LIN {X 0,Y 354.791,Z 411.293,A -85,B 0,C 180,E1 -13362.867,E2 -13362.867} C_VEL
LIN {X 0,Y 354.834,Z 411.311,A -85,B 0,C 180,E1 -13366.661,E2 -13366.661} C_VEL
LIN {X 0,Y 355.442,Z 414.83,A -85,B 0,C 180,E1 -13369.27,E2 -13369.27} C_VEL
LIN {X 0,Y 356.124,Z 419.11,A -85,B 0,C 180,E1 -13372.282,E2 -13372.282} C_VEL
LIN {X 0,Y 356.314,Z 421.652,A -85,B 0,C 180,E1 -13373.968,E2 -13373.968} C_VEL
LIN {X 0,Y 356.012,Z 425.546,A -85,B 0,C 180,E1 -13376.444,E2 -13376.444} C_VEL
LIN {X 0,Y 355.387,Z 431.994,A -85,B 0,C 180,E1 -13380.37,E2 -13380.37} C_VEL
LIN {X 0,Y 354.742,Z 438.379,A -85,B 0,C 180,E1 -13384.16,E2 -13384.16} C_VEL
LIN {X 0,Y 354.299,Z 444.723,A -85,B 0,C 180,E1 -13387.859,E2 -13387.859} C_VEL
LIN {X 0,Y 354.107,Z 447.535,A -85,B 0,C 180,E1 -13389.487,E2 -13389.487} C_VEL
LIN {X 0,Y 357.033,Z 461.918,A -85,B 0,C 180,E1 -13390.207,E2 -13390.207} C_VEL
LIN {X 0,Y 359.043,Z 475.173,A -85,B 0,C 180,E1 -13391.077,E2 -13391.077} C_VEL
LIN {X 0,Y 359.866,Z 484.104,A -85,B 0,C 180,E1 -13391.792,E2 -13391.792} C_VEL
LIN {X 0,Y 358.903,Z 495.118,A -85,B 0,C 180,E1 -13392.772,E2 -13392.772} C_VEL
LIN {X 0,Y 357.705,Z 506.362,A -85,B 0,C 180,E1 -13394.034,E2 -13394.034} C_VEL
LIN {X 0,Y 356.623,Z 516.327,A -85,B 0,C 180,E1 -13395.447,E2 -13395.447} C_VEL
LIN {X 0,Y 355.526,Z 525.99,A -85,B 0,C 180,E1 -13397.15,E2 -13397.15} C_VEL
LIN {X 0,Y 354.584,Z 533.681,A -85,B 0,C 180,E1 -13398.857,E2 -13398.857} C_VEL
LIN {X 0,Y 353.901,Z 540.779,A -85,B 0,C 180,E1 -13400.859,E2 -13400.859} C_VEL
LIN {X 0,Y 353.519,Z 545.502,A -85,B 0,C 180,E1 -13402.575,E2 -13402.575} C_VEL
LIN {X 0,Y 353.282,Z 549.111,A -85,B 0,C 180,E1 -13404.291,E2 -13404.291} C_VEL
LIN {X 0,Y 353.28,Z 550.976,A -85,B 0,C 180,E1 -13405.436,E2 -13405.436} C_VEL
LIN {X 0,Y 353.223,Z 552.372,A -85,B 0,C 180,E1 -13406.578,E2 -13406.578} C_VEL
LIN {X 0,Y 353.216,Z 553.978,A -85,B 0,C 180,E1 -13408.86,E2 -13408.86} C_VEL
LIN {X 0,Y 353.262,Z 554.194,A -85,B 0,C 180,E1 -13410,E2 -13410} C_VEL
LIN {X 0,Y 353.216,Z 553.974,A -85,B 0,C 180,E1 -13411.14,E2 -13411.14} C_VEL
LIN {X 0,Y 353.223,Z 552.364,A -85,B 0,C 180,E1 -13413.422,E2 -13413.422} C_VEL
LIN {X 0,Y 353.28,Z 550.964,A -85,B 0,C 180,E1 -13414.564,E2 -13414.564} C_VEL
LIN {X 0,Y 353.278,Z 548.719,A -85,B 0,C 180,E1 -13415.908,E2 -13415.908} C_VEL
LIN {X 0,Y 353.628,Z 544.039,A -85,B 0,C 180,E1 -13417.997,E2 -13417.997} C_VEL
LIN {X 0,Y 354.174,Z 537.919,A -85,B 0,C 180,E1 -13419.999,E2 -13419.999} C_VEL
LIN {X 0,Y 354.849,Z 531.235,A -85,B 0,C 180,E1 -13421.713,E2 -13421.713} C_VEL
LIN {X 0,Y 355.9,Z 522.95,A -85,B 0,C 180,E1 -13423.416,E2 -13423.416} C_VEL
LIN {X 0,Y 356.879,Z 514.454,A -85,B 0,C 180,E1 -13424.833,E2 -13424.833} C_VEL
LIN {X 0,Y 357.91,Z 503.953,A -85,B 0,C 180,E1 -13426.249,E2 -13426.249} C_VEL
LIN {X 0,Y 359.204,Z 492.142,A -85,B 0,C 180,E1 -13427.507,E2 -13427.507} C_VEL
LIN {X 0,Y 359.788,Z 482.88,A -85,B 0,C 180,E1 -13428.301,E2 -13428.301} C_VEL
LIN {X 0,Y 358.509,Z 471.103,A -85,B 0,C 180,E1 -13429.203,E2 -13429.203} C_VEL
LIN {X 0,Y 356.25,Z 457.832,A -85,B 0,C 180,E1 -13430.004,E2 -13430.004} C_VEL
LIN {X 0,Y 354.106,Z 447.512,A -85,B 0,C 180,E1 -13430.513,E2 -13430.513} C_VEL
LIN {X 0,Y 354.519,Z 441.111,A -85,B 0,C 180,E1 -13434.23,E2 -13434.23} C_VEL
LIN {X 0,Y 355.177,Z 434.088,A -85,B 0,C 180,E1 -13438.353,E2 -13438.353} C_VEL
LIN {X 0,Y 355.747,Z 428.287,A -85,B 0,C 180,E1 -13441.843,E2 -13441.843} C_VEL
LIN {X 0,Y 356.245,Z 423.356,A -85,B 0,C 180,E1 -13444.898,E2 -13444.898} C_VEL
LIN {X 0,Y 356.112,Z 418.838,A -85,B 0,C 180,E1 -13447.869,E2 -13447.869} C_VEL
LIN {X 0,Y 355.332,Z 414.036,A -85,B 0,C 180,E1 -13451.272,E2 -13451.272} C_VEL
LIN {X 0,Y 354.825,Z 411.291,A -85,B 0,C 180,E1 -13453.436,E2 -13453.436} C_VEL
LIN {X 0,Y 354.795,Z 411.288,A -85,B 0,C 180,E1 -13457.663,E2 -13457.663} C_VEL
LIN {X 0,Y 354.816,Z 411.287,A -85,B 0,C 180,E1 -13460.666,E2 -13460.666} C_VEL
LIN {X 0,Y 354.823,Z 411.285,A -85,B 0,C 180,E1 -13464.301,E2 -13464.301} C_VEL
LIN {X 0,Y 354.788,Z 411.288,A -85,B 0,C 180,E1 -13467.667,E2 -13467.667} C_VEL
LIN {X 0,Y 354.847,Z 411.28,A -85,B 0,C 180,E1 -13471.619,E2 -13471.619} C_VEL
LIN {X 0,Y 354.9,Z 411.275,A -85,B 0,C 180,E1 -13474.173,E2 -13474.173} C_VEL
LIN {X 0,Y 354.836,Z 411.282,A -85,B 0,C 180,E1 -13477.894,E2 -13477.894} C_VEL
LIN {X 0,Y 354.923,Z 411.271,A -85,B 0,C 180,E1 -13481.892,E2 -13481.892} C_VEL
LIN {X 0,Y 354.945,Z 411.27,A -85,B 0,C 180,E1 -13485.981,E2 -13485.981} C_VEL
LIN {X 0,Y 354.984,Z 411.264,A -85,B 0,C 180,E1 -13489.736,E2 -13489.736} C_VEL
LIN {X 0,Y 355.116,Z 411.25,A -85,B 0,C 180,E1 -13492.037,E2 -13492.037} C_VEL
LIN {X 0,Y 355.094,Z 411.256,A -85,B 0,C 180,E1 -13494.321,E2 -13494.321} C_VEL
LIN {X 0,Y 355.245,Z 411.232,A -85,B 0,C 180,E1 -13497.732,E2 -13497.732} C_VEL
LIN {X 0,Y 355.399,Z 411.215,A -85,B 0,C 180,E1 -13500,E2 -13500} C_VEL
LIN {X 0,Y 355.245,Z 411.236,A -85,B 0,C 180,E1 -13502.268,E2 -13502.268} C_VEL
LIN {X 0,Y 355.14,Z 411.244,A -85,B 0,C 180,E1 -13506.819,E2 -13506.819} C_VEL
LIN {X 0,Y 355.018,Z 411.259,A -85,B 0,C 180,E1 -13509.112,E2 -13509.112} C_VEL
LIN {X 0,Y 354.928,Z 411.271,A -85,B 0,C 180,E1 -13512.581,E2 -13512.581} C_VEL
LIN {X 0,Y 354.892,Z 411.279,A -85,B 0,C 180,E1 -13516.096,E2 -13516.096} C_VEL
LIN {X 0,Y 354.903,Z 411.274,A -85,B 0,C 180,E1 -13518.472,E2 -13518.472} C_VEL
LIN {X 0,Y 354.836,Z 411.285,A -85,B 0,C 180,E1 -13522.106,E2 -13522.106} C_VEL
LIN {X 0,Y 354.9,Z 411.279,A -85,B 0,C 180,E1 -13525.827,E2 -13525.827} C_VEL
LIN {X 0,Y 354.847,Z 411.286,A -85,B 0,C 180,E1 -13529.679,E2 -13529.679} C_VEL
LIN {X 0,Y 354.807,Z 411.29,A -85,B 0,C 180,E1 -13533.702,E2 -13533.702} C_VEL
LIN {X 0,Y 354.803,Z 411.286,A -85,B 0,C 180,E1 -13536.459,E2 -13536.459} C_VEL
LIN {X 0,Y 354.825,Z 411.289,A -85,B 0,C 180,E1 -13539.424,E2 -13539.424} C_VEL
LIN {X 0,Y 354.79,Z 411.289,A -85,B 0,C 180,E1 -13542.867,E2 -13542.867} C_VEL
LIN {X 0,Y 354.783,Z 411.289,A -85,B 0,C 180,E1 -13546.106,E2 -13546.106} C_VEL
LIN {X 0,Y 354.79,Z 411.293,A -85,B 0,C 180,E1 -13549.179,E2 -13549.179} C_VEL
LIN {X 0,Y 354.785,Z 411.293,A -85,B 0,C 180,E1 -13552.408,E2 -13552.408} C_VEL
LIN {X 0,Y 354.713,Z 411.303,A -85,B 0,C 180,E1 -13553.53,E2 -13553.53} C_VEL
LIN {X 0,Y 354.711,Z 414.22,A -85,B 0,C 180,E1 -13556.322,E2 -13556.322} C_VEL
LIN {X 0,Y 354.543,Z 417.115,A -85,B 0,C 180,E1 -13558.977,E2 -13558.977} C_VEL
LIN {X 0,Y 354.277,Z 421.498,A -85,B 0,C 180,E1 -13562.854,E2 -13562.854} C_VEL
LIN {X 0,Y 354.011,Z 425.915,A -85,B 0,C 180,E1 -13566.606,E2 -13566.606} C_VEL
LIN {X 0,Y 353.886,Z 429.701,A -85,B 0,C 180,E1 -13569.579,E2 -13569.579} C_VEL
LIN {X 0,Y 357.361,Z 443.1,A -85,B 0,C 180,E1 -13570.31,E2 -13570.31} C_VEL
LIN {X 0,Y 359.992,Z 455.598,A -85,B 0,C 180,E1 -13571.186,E2 -13571.186} C_VEL
LIN {X 0,Y 360.819,Z 460.678,A -85,B 0,C 180,E1 -13571.599,E2 -13571.599} C_VEL
LIN {X 0,Y 359.861,Z 471.979,A -85,B 0,C 180,E1 -13572.526,E2 -13572.526} C_VEL
LIN {X 0,Y 358.845,Z 482.845,A -85,B 0,C 180,E1 -13573.673,E2 -13573.673} C_VEL
LIN {X 0,Y 357.895,Z 492.362,A -85,B 0,C 180,E1 -13574.919,E2 -13574.919} C_VEL
LIN {X 0,Y 356.749,Z 501.204,A -85,B 0,C 180,E1 -13576.326,E2 -13576.326} C_VEL
LIN {X 0,Y 355.757,Z 509.824,A -85,B 0,C 180,E1 -13578.028,E2 -13578.028} C_VEL
LIN {X 0,Y 354.916,Z 516.695,A -85,B 0,C 180,E1 -13579.734,E2 -13579.734} C_VEL
LIN {X 0,Y 354.205,Z 522.198,A -85,B 0,C 180,E1 -13581.442,E2 -13581.442} C_VEL
LIN {X 0,Y 353.808,Z 526.852,A -85,B 0,C 180,E1 -13583.313,E2 -13583.313} C_VEL
LIN {X 0,Y 353.498,Z 530.652,A -85,B 0,C 180,E1 -13585.439,E2 -13585.439} C_VEL
LIN {X 0,Y 353.339,Z 532.051,A -85,B 0,C 180,E1 -13586.579,E2 -13586.579} C_VEL
LIN {X 0,Y 353.256,Z 533.656,A -85,B 0,C 180,E1 -13588.86,E2 -13588.86} C_VEL
LIN {X 0,Y 353.265,Z 533.887,A -85,B 0,C 180,E1 -13590,E2 -13590} C_VEL
LIN {X 0,Y 353.256,Z 533.698,A -85,B 0,C 180,E1 -13591.14,E2 -13591.14} C_VEL
LIN {X 0,Y 353.334,Z 532.147,A -85,B 0,C 180,E1 -13593.421,E2 -13593.421} C_VEL
LIN {X 0,Y 353.491,Z 530.789,A -85,B 0,C 180,E1 -13594.561,E2 -13594.561} C_VEL
LIN {X 0,Y 353.762,Z 527.213,A -85,B 0,C 180,E1 -13596.622,E2 -13596.622} C_VEL
LIN {X 0,Y 354.201,Z 522.482,A -85,B 0,C 180,E1 -13598.558,E2 -13598.558} C_VEL
LIN {X 0,Y 354.994,Z 516.044,A -85,B 0,C 180,E1 -13600.552,E2 -13600.552} C_VEL
LIN {X 0,Y 355.783,Z 508.972,A -85,B 0,C 180,E1 -13602.26,E2 -13602.26} C_VEL
LIN {X 0,Y 356.925,Z 500.154,A -85,B 0,C 180,E1 -13603.958,E2 -13603.958} C_VEL
LIN {X 0,Y 358.06,Z 491.103,A -85,B 0,C 180,E1 -13605.366,E2 -13605.366} C_VEL
LIN {X 0,Y 358.921,Z 481.466,A -85,B 0,C 180,E1 -13606.597,E2 -13606.597} C_VEL
LIN {X 0,Y 360.084,Z 469.933,A -85,B 0,C 180,E1 -13607.756,E2 -13607.756} C_VEL
LIN {X 0,Y 360.798,Z 460.4,A -85,B 0,C 180,E1 -13608.526,E2 -13608.526} C_VEL
LIN {X 0,Y 358.493,Z 448.093,A -85,B 0,C 180,E1 -13609.468,E2 -13609.468} C_VEL
LIN {X 0,Y 355.478,Z 435.673,A -85,B 0,C 180,E1 -13610.23,E2 -13610.23} C_VEL
LIN {X 0,Y 353.87,Z 429.539,A -85,B 0,C 180,E1 -13610.558,E2 -13610.558} C_VEL
LIN {X 0,Y 354.103,Z 424.577,A -85,B 0,C 180,E1 -13614.633,E2 -13614.633} C_VEL
LIN {X 0,Y 354.281,Z 421.637,A -85,B 0,C 180,E1 -13617.146,E2 -13617.146} C_VEL
LIN {X 0,Y 354.538,Z 417.231,A -85,B 0,C 180,E1 -13621.024,E2 -13621.024} C_VEL
LIN {X 0,Y 354.713,Z 414.326,A -85,B 0,C 180,E1 -13623.695,E2 -13623.695} C_VEL
LIN {X 0,Y 354.754,Z 411.408,A -85,B 0,C 180,E1 -13626.465,E2 -13626.465} C_VEL
LIN {X 0,Y 354.793,Z 411.291,A -85,B 0,C 180,E1 -13627.872,E2 -13627.872} C_VEL
LIN {X 0,Y 354.144,Z 411.374,A -85,B 0,C 180,E1 -13628.819,E2 -13628.819} C_VEL
LIN {X 0,Y 351.269,Z 411.728,A -85,B 0,C 180,E1 -13630.359,E2 -13630.359} C_VEL
LIN {X 0,Y 348.827,Z 412.03,A -85,B 0,C 180,E1 -13631.604,E2 -13631.604} C_VEL
LIN {X 0,Y 347.79,Z 412.163,A -85,B 0,C 180,E1 -13632.569,E2 -13632.569} C_VEL
LIN {X 0,Y 347.713,Z 412.167,A -85,B 0,C 180,E1 -13632.896,E2 -13632.896} C_VEL
LIN {X 0,Y 347.768,Z 412.165,A -85,B 0,C 180,E1 -13635.017,E2 -13635.017} C_VEL
LIN {X 0,Y 347.753,Z 412.168,A -85,B 0,C 180,E1 -13638.397,E2 -13638.397} C_VEL
LIN {X 0,Y 347.779,Z 412.162,A -85,B 0,C 180,E1 -13642.011,E2 -13642.011} C_VEL
LIN {X 0,Y 347.747,Z 412.165,A -85,B 0,C 180,E1 -13645.536,E2 -13645.536} C_VEL
LIN {X 0,Y 347.763,Z 412.163,A -85,B 0,C 180,E1 -13649.653,E2 -13649.653} C_VEL
LIN {X 0,Y 347.833,Z 412.154,A -85,B 0,C 180,E1 -13653.608,E2 -13653.608} C_VEL
LIN {X 0,Y 347.791,Z 412.164,A -85,B 0,C 180,E1 -13656.162,E2 -13656.162} C_VEL
LIN {X 0,Y 347.815,Z 412.159,A -85,B 0,C 180,E1 -13659.909,E2 -13659.909} C_VEL
LIN {X 0,Y 347.869,Z 412.154,A -85,B 0,C 180,E1 -13662.359,E2 -13662.359} C_VEL
LIN {X 0,Y 347.9,Z 412.15,A -85,B 0,C 180,E1 -13665.971,E2 -13665.971} C_VEL
LIN {X 0,Y 347.932,Z 412.143,A -85,B 0,C 180,E1 -13669.526,E2 -13669.526} C_VEL
LIN {X 0,Y 348.077,Z 412.128,A -85,B 0,C 180,E1 -13671.875,E2 -13671.875} C_VEL
LIN {X 0,Y 348.07,Z 412.128,A -85,B 0,C 180,E1 -13674.206,E2 -13674.206} C_VEL
LIN {X 0,Y 348.209,Z 412.111,A -85,B 0,C 180,E1 -13677.686,E2 -13677.686} C_VEL
LIN {X 0,Y 348.348,Z 412.094,A -85,B 0,C 180,E1 -13680,E2 -13680} C_VEL
LIN {X 0,Y 348.209,Z 412.108,A -85,B 0,C 180,E1 -13682.313,E2 -13682.313} C_VEL
LIN {X 0,Y 348.11,Z 412.12,A -85,B 0,C 180,E1 -13686.958,E2 -13686.958} C_VEL
LIN {X 0,Y 347.972,Z 412.14,A -85,B 0,C 180,E1 -13689.298,E2 -13689.298} C_VEL
LIN {X 0,Y 347.897,Z 412.147,A -85,B 0,C 180,E1 -13692.839,E2 -13692.839} C_VEL
LIN {X 0,Y 347.842,Z 412.153,A -85,B 0,C 180,E1 -13696.431,E2 -13696.431} C_VEL
LIN {X 0,Y 347.854,Z 412.153,A -85,B 0,C 180,E1 -13698.86,E2 -13698.86} C_VEL
LIN {X 0,Y 347.777,Z 412.161,A -85,B 0,C 180,E1 -13702.579,E2 -13702.579} C_VEL
LIN {X 0,Y 347.815,Z 412.16,A -85,B 0,C 180,E1 -13705.108,E2 -13705.108} C_VEL
LIN {X 0,Y 347.81,Z 412.159,A -85,B 0,C 180,E1 -13707.694,E2 -13707.694} C_VEL
LIN {X 0,Y 347.751,Z 412.165,A -85,B 0,C 180,E1 -13710.348,E2 -13710.348} C_VEL
LIN {X 0,Y 347.75,Z 412.164,A -85,B 0,C 180,E1 -13714.044,E2 -13714.044} C_VEL
LIN {X 0,Y 347.765,Z 412.166,A -85,B 0,C 180,E1 -13717.321,E2 -13717.321} C_VEL
LIN {X 0,Y 347.735,Z 412.168,A -85,B 0,C 180,E1 -13720.297,E2 -13720.297} C_VEL
LIN {X 0,Y 347.729,Z 412.172,A -85,B 0,C 180,E1 -13723.407,E2 -13723.407} C_VEL
LIN {X 0,Y 347.776,Z 412.228,A -85,B 0,C 180,E1 -13726.346,E2 -13726.346} C_VEL
LIN {X 0,Y 348.609,Z 417.085,A -85,B 0,C 180,E1 -13730.004,E2 -13730.004} C_VEL
LIN {X 0,Y 349.215,Z 421.12,A -85,B 0,C 180,E1 -13732.86,E2 -13732.86} C_VEL
LIN {X 0,Y 349.252,Z 424.325,A -85,B 0,C 180,E1 -13735.005,E2 -13735.005} C_VEL
LIN {X 0,Y 348.559,Z 430.751,A -85,B 0,C 180,E1 -13739.059,E2 -13739.059} C_VEL
LIN {X 0,Y 347.892,Z 436.757,A -85,B 0,C 180,E1 -13742.732,E2 -13742.732} C_VEL
LIN {X 0,Y 347.419,Z 442.433,A -85,B 0,C 180,E1 -13746.135,E2 -13746.135} C_VEL
LIN {X 0,Y 347.068,Z 447.32,A -85,B 0,C 180,E1 -13749.051,E2 -13749.051} C_VEL
LIN {X 0,Y 350.077,Z 461.716,A -85,B 0,C 180,E1 -13749.797,E2 -13749.797} C_VEL
LIN {X 0,Y 352.083,Z 474.968,A -85,B 0,C 180,E1 -13750.688,E2 -13750.688} C_VEL
LIN {X 0,Y 353.013,Z 485.675,A -85,B 0,C 180,E1 -13751.576,E2 -13751.576} C_VEL
LIN {X 0,Y 351.986,Z 496.339,A -85,B 0,C 180,E1 -13752.572,E2 -13752.572} C_VEL
LIN {X 0,Y 350.714,Z 507.306,A -85,B 0,C 180,E1 -13753.867,E2 -13753.867} C_VEL
LIN {X 0,Y 349.74,Z 516.125,A -85,B 0,C 180,E1 -13755.155,E2 -13755.155} C_VEL
LIN {X 0,Y 348.571,Z 525.787,A -85,B 0,C 180,E1 -13756.89,E2 -13756.89} C_VEL
LIN {X 0,Y 347.564,Z 533.477,A -85,B 0,C 180,E1 -13758.629,E2 -13758.629} C_VEL
LIN {X 0,Y 346.871,Z 540.575,A -85,B 0,C 180,E1 -13760.672,E2 -13760.672} C_VEL
LIN {X 0,Y 346.47,Z 545.298,A -85,B 0,C 180,E1 -13762.423,E2 -13762.423} C_VEL
LIN {X 0,Y 346.201,Z 548.907,A -85,B 0,C 180,E1 -13764.174,E2 -13764.174} C_VEL
LIN {X 0,Y 346.175,Z 550.771,A -85,B 0,C 180,E1 -13765.342,E2 -13765.342} C_VEL
LIN {X 0,Y 346.147,Z 552.169,A -85,B 0,C 180,E1 -13766.508,E2 -13766.508} C_VEL
LIN {X 0,Y 346.116,Z 553.774,A -85,B 0,C 180,E1 -13768.836,E2 -13768.836} C_VEL
LIN {X 0,Y 346.165,Z 553.99,A -85,B 0,C 180,E1 -13770,E2 -13770} C_VEL
LIN {X 0,Y 346.116,Z 553.769,A -85,B 0,C 180,E1 -13771.163,E2 -13771.163} C_VEL
LIN {X 0,Y 346.147,Z 552.16,A -85,B 0,C 180,E1 -13773.492,E2 -13773.492} C_VEL
LIN {X 0,Y 346.175,Z 550.759,A -85,B 0,C 180,E1 -13774.658,E2 -13774.658} C_VEL
LIN {X 0,Y 346.241,Z 547.814,A -85,B 0,C 180,E1 -13776.409,E2 -13776.409} C_VEL
LIN {X 0,Y 346.571,Z 543.833,A -85,B 0,C 180,E1 -13778.161,E2 -13778.161} C_VEL
LIN {X 0,Y 347.146,Z 537.713,A -85,B 0,C 180,E1 -13780.203,E2 -13780.203} C_VEL
LIN {X 0,Y 347.847,Z 531.028,A -85,B 0,C 180,E1 -13781.952,E2 -13781.952} C_VEL
LIN {X 0,Y 348.972,Z 522.743,A -85,B 0,C 180,E1 -13783.688,E2 -13783.688} C_VEL
LIN {X 0,Y 350.006,Z 514.247,A -85,B 0,C 180,E1 -13785.131,E2 -13785.131} C_VEL
LIN {X 0,Y 351.061,Z 503.745,A -85,B 0,C 180,E1 -13786.575,E2 -13786.575} C_VEL
LIN {X 0,Y 352.428,Z 491.934,A -85,B 0,C 180,E1 -13787.855,E2 -13787.855} C_VEL
LIN {X 0,Y 352.932,Z 483.739,A -85,B 0,C 180,E1 -13788.579,E2 -13788.579} C_VEL
LIN {X 0,Y 351.559,Z 470.884,A -85,B 0,C 180,E1 -13789.598,E2 -13789.598} C_VEL
LIN {X 0,Y 349.239,Z 457.562,A -85,B 0,C 180,E1 -13790.426,E2 -13790.426} C_VEL
LIN {X 0,Y 347.081,Z 447.329,A -85,B 0,C 180,E1 -13790.928,E2 -13790.928} C_VEL
LIN {X 0,Y 347.503,Z 441.37,A -85,B 0,C 180,E1 -13794.481,E2 -13794.481} C_VEL
LIN {X 0,Y 348.104,Z 434.977,A -85,B 0,C 180,E1 -13798.324,E2 -13798.324} C_VEL
LIN {X 0,Y 348.658,Z 429.637,A -85,B 0,C 180,E1 -13801.607,E2 -13801.607} C_VEL
LIN {X 0,Y 349.221,Z 424.267,A -85,B 0,C 180,E1 -13804.998,E2 -13804.998} C_VEL
LIN {X 0,Y 349.2,Z 421.046,A -85,B 0,C 180,E1 -13807.141,E2 -13807.141} C_VEL
LIN {X 0,Y 348.571,Z 416.771,A -85,B 0,C 180,E1 -13810.18,E2 -13810.18} C_VEL
LIN {X 0,Y 347.779,Z 412.169,A -85,B 0,C 180,E1 -13813.71,E2 -13813.71} C_VEL
LIN {X 0,Y 347.726,Z 412.172,A -85,B 0,C 180,E1 -13816.686,E2 -13816.686} C_VEL
LIN {X 0,Y 347.748,Z 412.166,A -85,B 0,C 180,E1 -13820.173,E2 -13820.173} C_VEL
LIN {X 0,Y 347.764,Z 412.167,A -85,B 0,C 180,E1 -13822.679,E2 -13822.679} C_VEL
LIN {X 0,Y 347.749,Z 412.165,A -85,B 0,C 180,E1 -13825.956,E2 -13825.956} C_VEL
LIN {X 0,Y 347.75,Z 412.165,A -85,B 0,C 180,E1 -13829.652,E2 -13829.652} C_VEL
LIN {X 0,Y 347.832,Z 412.154,A -85,B 0,C 180,E1 -13833.608,E2 -13833.608} C_VEL
LIN {X 0,Y 347.79,Z 412.161,A -85,B 0,C 180,E1 -13836.162,E2 -13836.162} C_VEL
LIN {X 0,Y 347.814,Z 412.157,A -85,B 0,C 180,E1 -13839.909,E2 -13839.909} C_VEL
LIN {X 0,Y 347.867,Z 412.154,A -85,B 0,C 180,E1 -13842.359,E2 -13842.359} C_VEL
LIN {X 0,Y 347.899,Z 412.147,A -85,B 0,C 180,E1 -13845.971,E2 -13845.971} C_VEL
LIN {X 0,Y 347.935,Z 412.142,A -85,B 0,C 180,E1 -13849.526,E2 -13849.526} C_VEL
LIN {X 0,Y 348.076,Z 412.125,A -85,B 0,C 180,E1 -13851.875,E2 -13851.875} C_VEL
LIN {X 0,Y 348.069,Z 412.129,A -85,B 0,C 180,E1 -13854.206,E2 -13854.206} C_VEL
LIN {X 0,Y 348.208,Z 412.108,A -85,B 0,C 180,E1 -13857.687,E2 -13857.687} C_VEL
LIN {X 0,Y 348.369,Z 412.091,A -85,B 0,C 180,E1 -13860,E2 -13860} C_VEL
LIN {X 0,Y 348.207,Z 412.112,A -85,B 0,C 180,E1 -13862.314,E2 -13862.314} C_VEL
LIN {X 0,Y 348.108,Z 412.12,A -85,B 0,C 180,E1 -13866.958,E2 -13866.958} C_VEL
LIN {X 0,Y 347.971,Z 412.137,A -85,B 0,C 180,E1 -13869.299,E2 -13869.299} C_VEL
LIN {X 0,Y 347.896,Z 412.146,A -85,B 0,C 180,E1 -13872.839,E2 -13872.839} C_VEL
LIN {X 0,Y 347.841,Z 412.155,A -85,B 0,C 180,E1 -13876.431,E2 -13876.431} C_VEL
LIN {X 0,Y 347.852,Z 412.151,A -85,B 0,C 180,E1 -13878.861,E2 -13878.861} C_VEL
LIN {X 0,Y 347.776,Z 412.161,A -85,B 0,C 180,E1 -13882.579,E2 -13882.579} C_VEL
LIN {X 0,Y 347.813,Z 412.157,A -85,B 0,C 180,E1 -13885.108,E2 -13885.108} C_VEL
LIN {X 0,Y 347.809,Z 412.163,A -85,B 0,C 180,E1 -13887.694,E2 -13887.694} C_VEL
LIN {X 0,Y 347.762,Z 412.163,A -85,B 0,C 180,E1 -13890.347,E2 -13890.347} C_VEL
LIN {X 0,Y 347.746,Z 412.165,A -85,B 0,C 180,E1 -13894.464,E2 -13894.464} C_VEL
LIN {X 0,Y 347.779,Z 412.163,A -85,B 0,C 180,E1 -13897.99,E2 -13897.99} C_VEL
LIN {X 0,Y 347.752,Z 412.166,A -85,B 0,C 180,E1 -13901.83,E2 -13901.83} C_VEL
LIN {X 0,Y 347.768,Z 412.165,A -85,B 0,C 180,E1 -13905.017,E2 -13905.017} C_VEL
LIN {X 0,Y 347.752,Z 412.165,A -85,B 0,C 180,E1 -13908.397,E2 -13908.397} C_VEL
LIN {X 0,Y 347.762,Z 412.168,A -85,B 0,C 180,E1 -13912.014,E2 -13912.014} C_VEL
LIN {X 0,Y 347.704,Z 412.733,A -85,B 0,C 180,E1 -13913.95,E2 -13913.95} C_VEL
LIN {X 0,Y 347.616,Z 415.827,A -85,B 0,C 180,E1 -13916.915,E2 -13916.915} C_VEL
LIN {X 0,Y 347.376,Z 419.657,A -85,B 0,C 180,E1 -13920.455,E2 -13920.455} C_VEL
LIN {X 0,Y 347.181,Z 423.157,A -85,B 0,C 180,E1 -13923.555,E2 -13923.555} C_VEL
LIN {X 0,Y 347.024,Z 426.109,A -85,B 0,C 180,E1 -13926.106,E2 -13926.106} C_VEL
LIN {X 0,Y 346.82,Z 429.857,A -85,B 0,C 180,E1 -13929.141,E2 -13929.141} C_VEL
LIN {X 0,Y 350.335,Z 443.072,A -85,B 0,C 180,E1 -13929.886,E2 -13929.886} C_VEL
LIN {X 0,Y 352.73,Z 454.179,A -85,B 0,C 180,E1 -13930.673,E2 -13930.673} C_VEL
LIN {X 0,Y 354.008,Z 462.099,A -85,B 0,C 180,E1 -13931.324,E2 -13931.324} C_VEL
LIN {X 0,Y 352.923,Z 473.628,A -85,B 0,C 180,E1 -13932.321,E2 -13932.321} C_VEL
LIN {X 0,Y 351.983,Z 483.625,A -85,B 0,C 180,E1 -13933.418,E2 -13933.418} C_VEL
LIN {X 0,Y 351.056,Z 492.569,A -85,B 0,C 180,E1 -13934.618,E2 -13934.618} C_VEL
LIN {X 0,Y 349.867,Z 501.411,A -85,B 0,C 180,E1 -13936.051,E2 -13936.051} C_VEL
LIN {X 0,Y 348.822,Z 510.03,A -85,B 0,C 180,E1 -13937.787,E2 -13937.787} C_VEL
LIN {X 0,Y 347.936,Z 516.901,A -85,B 0,C 180,E1 -13939.526,E2 -13939.526} C_VEL
LIN {X 0,Y 347.18,Z 522.403,A -85,B 0,C 180,E1 -13941.268,E2 -13941.268} C_VEL
LIN {X 0,Y 346.731,Z 527.351,A -85,B 0,C 180,E1 -13943.316,E2 -13943.316} C_VEL
LIN {X 0,Y 346.44,Z 530.856,A -85,B 0,C 180,E1 -13945.346,E2 -13945.346} C_VEL
LIN {X 0,Y 346.264,Z 532.255,A -85,B 0,C 180,E1 -13946.509,E2 -13946.509} C_VEL
LIN {X 0,Y 346.16,Z 533.86,A -85,B 0,C 180,E1 -13948.837,E2 -13948.837} C_VEL
LIN {X 0,Y 346.168,Z 534.091,A -85,B 0,C 180,E1 -13950,E2 -13950} C_VEL
LIN {X 0,Y 346.159,Z 533.901,A -85,B 0,C 180,E1 -13951.163,E2 -13951.163} C_VEL
LIN {X 0,Y 346.259,Z 532.35,A -85,B 0,C 180,E1 -13953.491,E2 -13953.491} C_VEL
LIN {X 0,Y 346.433,Z 530.992,A -85,B 0,C 180,E1 -13954.655,E2 -13954.655} C_VEL
LIN {X 0,Y 346.682,Z 527.715,A -85,B 0,C 180,E1 -13956.616,E2 -13956.616} C_VEL
LIN {X 0,Y 347.176,Z 522.685,A -85,B 0,C 180,E1 -13958.733,E2 -13958.733} C_VEL
LIN {X 0,Y 347.984,Z 516.247,A -85,B 0,C 180,E1 -13960.767,E2 -13960.767} C_VEL
LIN {X 0,Y 348.843,Z 509.174,A -85,B 0,C 180,E1 -13962.508,E2 -13962.508} C_VEL
LIN {X 0,Y 350.052,Z 500.354,A -85,B 0,C 180,E1 -13964.238,E2 -13964.238} C_VEL
LIN {X 0,Y 351.212,Z 491.419,A -85,B 0,C 180,E1 -13965.655,E2 -13965.655} C_VEL
LIN {X 0,Y 352.132,Z 481.665,A -85,B 0,C 180,E1 -13966.927,E2 -13966.927} C_VEL
LIN {X 0,Y 353.346,Z 470.131,A -85,B 0,C 180,E1 -13968.106,E2 -13968.106} C_VEL
LIN {X 0,Y 353.937,Z 460.879,A -85,B 0,C 180,E1 -13968.878,E2 -13968.878} C_VEL
LIN {X 0,Y 351.503,Z 448.297,A -85,B 0,C 180,E1 -13969.871,E2 -13969.871} C_VEL
LIN {X 0,Y 348.415,Z 435.647,A -85,B 0,C 180,E1 -13970.668,E2 -13970.668} C_VEL
LIN {X 0,Y 346.819,Z 429.759,A -85,B 0,C 180,E1 -13970.983,E2 -13970.983} C_VEL
LIN {X 0,Y 347.033,Z 425.753,A -85,B 0,C 180,E1 -13974.31,E2 -13974.31} C_VEL
LIN {X 0,Y 347.264,Z 421.813,A -85,B 0,C 180,E1 -13977.741,E2 -13977.741} C_VEL
LIN {X 0,Y 347.544,Z 417.398,A -85,B 0,C 180,E1 -13981.72,E2 -13981.72} C_VEL
LIN {X 0,Y 347.68,Z 414.472,A -85,B 0,C 180,E1 -13984.471,E2 -13984.471} C_VEL
LIN {X 0,Y 347.751,Z 412.838,A -85,B 0,C 180,E1 -13986.06,E2 -13986.06} C_VEL
LIN {X 0,Y 347.74,Z 412.17,A -85,B 0,C 180,E1 -13987.324,E2 -13987.324} C_VEL
LIN {X 0,Y 347.735,Z 412.168,A -85,B 0,C 180,E1 -13990.297,E2 -13990.297} C_VEL
LIN {X 0,Y 347.713,Z 412.167,A -85,B 0,C 180,E1 -13992.896,E2 -13992.896} C_VEL
LIN {X 0,Y 347.074,Z 412.25,A -85,B 0,C 180,E1 -13993.863,E2 -13993.863} C_VEL
LIN {X 0,Y 344.258,Z 412.601,A -85,B 0,C 180,E1 -13995.437,E2 -13995.437} C_VEL
LIN {X 0,Y 341.847,Z 412.906,A -85,B 0,C 180,E1 -13996.711,E2 -13996.711} C_VEL
LIN {X 0,Y 340.793,Z 413.032,A -85,B 0,C 180,E1 -13997.696,E2 -13997.696} C_VEL
LIN {X 0,Y 340.697,Z 413.044,A -85,B 0,C 180,E1 -13998.03,E2 -13998.03} C_VEL
LIN {X 0,Y 340.738,Z 413.038,A -85,B 0,C 180,E1 -14001.773,E2 -14001.773} C_VEL
LIN {X 0,Y 340.725,Z 413.04,A -85,B 0,C 180,E1 -14005.595,E2 -14005.595} C_VEL
LIN {X 0,Y 340.771,Z 413.036,A -85,B 0,C 180,E1 -14010.021,E2 -14010.021} C_VEL
LIN {X 0,Y 340.806,Z 413.03,A -85,B 0,C 180,E1 -14013.02,E2 -14013.02} C_VEL
LIN {X 0,Y 340.759,Z 413.036,A -85,B 0,C 180,E1 -14015.638,E2 -14015.638} C_VEL
LIN {X 0,Y 340.748,Z 413.037,A -85,B 0,C 180,E1 -14019.474,E2 -14019.474} C_VEL
LIN {X 0,Y 340.86,Z 413.027,A -85,B 0,C 180,E1 -14021.984,E2 -14021.984} C_VEL
LIN {X 0,Y 340.872,Z 413.023,A -85,B 0,C 180,E1 -14025.705,E2 -14025.705} C_VEL
LIN {X 0,Y 340.874,Z 413.021,A -85,B 0,C 180,E1 -14029.306,E2 -14029.306} C_VEL
LIN {X 0,Y 341.079,Z 412.996,A -85,B 0,C 180,E1 -14032.898,E2 -14032.898} C_VEL
LIN {X 0,Y 341.17,Z 412.988,A -85,B 0,C 180,E1 -14037.639,E2 -14037.639} C_VEL
LIN {X 0,Y 341.298,Z 412.973,A -85,B 0,C 180,E1 -14040,E2 -14040} C_VEL
LIN {X 0,Y 341.171,Z 412.985,A -85,B 0,C 180,E1 -14042.361,E2 -14042.361} C_VEL
LIN {X 0,Y 341.079,Z 412.997,A -85,B 0,C 180,E1 -14047.102,E2 -14047.102} C_VEL
LIN {X 0,Y 340.878,Z 413.02,A -85,B 0,C 180,E1 -14050.694,E2 -14050.694} C_VEL
LIN {X 0,Y 340.865,Z 413.022,A -85,B 0,C 180,E1 -14054.325,E2 -14054.325} C_VEL
LIN {X 0,Y 340.839,Z 413.025,A -85,B 0,C 180,E1 -14058.466,E2 -14058.466} C_VEL
LIN {X 0,Y 340.756,Z 413.037,A -85,B 0,C 180,E1 -14061.857,E2 -14061.857} C_VEL
LIN {X 0,Y 340.775,Z 413.036,A -85,B 0,C 180,E1 -14065.664,E2 -14065.664} C_VEL
LIN {X 0,Y 340.731,Z 413.039,A -85,B 0,C 180,E1 -14068.321,E2 -14068.321} C_VEL
LIN {X 0,Y 340.7,Z 413.047,A -85,B 0,C 180,E1 -14071.045,E2 -14071.045} C_VEL
LIN {X 0,Y 340.72,Z 413.044,A -85,B 0,C 180,E1 -14075.279,E2 -14075.279} C_VEL
LIN {X 0,Y 340.712,Z 413.042,A -85,B 0,C 180,E1 -14078.386,E2 -14078.386} C_VEL
LIN {X 0,Y 340.701,Z 413.044,A -85,B 0,C 180,E1 -14082.045,E2 -14082.045} C_VEL
LIN {X 0,Y 340.734,Z 413.105,A -85,B 0,C 180,E1 -14085.999,E2 -14085.999} C_VEL
LIN {X 0,Y 341.519,Z 417.738,A -85,B 0,C 180,E1 -14089.589,E2 -14089.589} C_VEL
LIN {X 0,Y 342.026,Z 420.957,A -85,B 0,C 180,E1 -14091.943,E2 -14091.943} C_VEL
LIN {X 0,Y 342.282,Z 424.177,A -85,B 0,C 180,E1 -14094.184,E2 -14094.184} C_VEL
LIN {X 0,Y 341.96,Z 427.368,A -85,B 0,C 180,E1 -14096.295,E2 -14096.295} C_VEL
LIN {X 0,Y 341.359,Z 432.936,A -85,B 0,C 180,E1 -14099.85,E2 -14099.85} C_VEL
LIN {X 0,Y 340.768,Z 438.008,A -85,B 0,C 180,E1 -14103.017,E2 -14103.017} C_VEL
LIN {X 0,Y 340.274,Z 444.316,A -85,B 0,C 180,E1 -14106.894,E2 -14106.894} C_VEL
LIN {X 0,Y 340.051,Z 447.16,A -85,B 0,C 180,E1 -14108.614,E2 -14108.614} C_VEL
LIN {X 0,Y 342.859,Z 460.305,A -85,B 0,C 180,E1 -14109.291,E2 -14109.291} C_VEL
LIN {X 0,Y 344.865,Z 472.572,A -85,B 0,C 180,E1 -14110.118,E2 -14110.118} C_VEL
LIN {X 0,Y 346.041,Z 483.696,A -85,B 0,C 180,E1 -14111.037,E2 -14111.037} C_VEL
LIN {X 0,Y 346.003,Z 488.743,A -85,B 0,C 180,E1 -14111.496,E2 -14111.496} C_VEL
LIN {X 0,Y 344.74,Z 500.038,A -85,B 0,C 180,E1 -14112.653,E2 -14112.653} C_VEL
LIN {X 0,Y 343.572,Z 509.764,A -85,B 0,C 180,E1 -14113.901,E2 -14113.901} C_VEL
LIN {X 0,Y 342.426,Z 519.386,A -85,B 0,C 180,E1 -14115.438,E2 -14115.438} C_VEL
LIN {X 0,Y 341.262,Z 528.321,A -85,B 0,C 180,E1 -14117.209,E2 -14117.209} C_VEL
LIN {X 0,Y 340.363,Z 535.514,A -85,B 0,C 180,E1 -14118.989,E2 -14118.989} C_VEL
LIN {X 0,Y 339.683,Z 542.068,A -85,B 0,C 180,E1 -14121.073,E2 -14121.073} C_VEL
LIN {X 0,Y 339.275,Z 546.406,A -85,B 0,C 180,E1 -14122.86,E2 -14122.86} C_VEL
LIN {X 0,Y 339.112,Z 548.876,A -85,B 0,C 180,E1 -14124.148,E2 -14124.148} C_VEL
LIN {X 0,Y 339.076,Z 550.567,A -85,B 0,C 180,E1 -14125.244,E2 -14125.244} C_VEL
LIN {X 0,Y 339.071,Z 551.965,A -85,B 0,C 180,E1 -14126.435,E2 -14126.435} C_VEL
LIN {X 0,Y 339.018,Z 553.57,A -85,B 0,C 180,E1 -14128.812,E2 -14128.812} C_VEL
LIN {X 0,Y 339.068,Z 553.786,A -85,B 0,C 180,E1 -14130,E2 -14130} C_VEL
LIN {X 0,Y 339.018,Z 553.565,A -85,B 0,C 180,E1 -14131.188,E2 -14131.188} C_VEL
LIN {X 0,Y 339.071,Z 551.956,A -85,B 0,C 180,E1 -14133.565,E2 -14133.565} C_VEL
LIN {X 0,Y 339.076,Z 550.553,A -85,B 0,C 180,E1 -14134.756,E2 -14134.756} C_VEL
LIN {X 0,Y 339.166,Z 547.608,A -85,B 0,C 180,E1 -14136.544,E2 -14136.544} C_VEL
LIN {X 0,Y 339.531,Z 543.627,A -85,B 0,C 180,E1 -14138.331,E2 -14138.331} C_VEL
LIN {X 0,Y 340.123,Z 537.506,A -85,B 0,C 180,E1 -14140.416,E2 -14140.416} C_VEL
LIN {X 0,Y 340.87,Z 530.821,A -85,B 0,C 180,E1 -14142.2,E2 -14142.2} C_VEL
LIN {X 0,Y 342.05,Z 522.536,A -85,B 0,C 180,E1 -14143.971,E2 -14143.971} C_VEL
LIN {X 0,Y 343.244,Z 513.005,A -85,B 0,C 180,E1 -14145.599,E2 -14145.599} C_VEL
LIN {X 0,Y 344.394,Z 502.36,A -85,B 0,C 180,E1 -14147.058,E2 -14147.058} C_VEL
LIN {X 0,Y 345.661,Z 491.725,A -85,B 0,C 180,E1 -14148.216,E2 -14148.216} C_VEL
LIN {X 0,Y 346.128,Z 485.303,A -85,B 0,C 180,E1 -14148.804,E2 -14148.804} C_VEL
LIN {X 0,Y 344.938,Z 473.028,A -85,B 0,C 180,E1 -14149.83,E2 -14149.83} C_VEL
LIN {X 0,Y 342.82,Z 460.171,A -85,B 0,C 180,E1 -14150.702,E2 -14150.702} C_VEL
LIN {X 0,Y 340.054,Z 447.111,A -85,B 0,C 180,E1 -14151.393,E2 -14151.393} C_VEL
LIN {X 0,Y 340.465,Z 441.648,A -85,B 0,C 180,E1 -14154.733,E2 -14154.733} C_VEL
LIN {X 0,Y 341.159,Z 434.793,A -85,B 0,C 180,E1 -14158.954,E2 -14158.954} C_VEL
LIN {X 0,Y 341.759,Z 429.154,A -85,B 0,C 180,E1 -14162.527,E2 -14162.527} C_VEL
LIN {X 0,Y 342.209,Z 425.186,A -85,B 0,C 180,E1 -14165.102,E2 -14165.102} C_VEL
LIN {X 0,Y 342.034,Z 420.901,A -85,B 0,C 180,E1 -14168.056,E2 -14168.056} C_VEL
LIN {X 0,Y 341.367,Z 416.62,A -85,B 0,C 180,E1 -14171.209,E2 -14171.209} C_VEL
LIN {X 0,Y 340.711,Z 413.047,A -85,B 0,C 180,E1 -14174.115,E2 -14174.115} C_VEL
LIN {X 0,Y 340.7,Z 413.044,A -85,B 0,C 180,E1 -14177.954,E2 -14177.954} C_VEL
LIN {X 0,Y 340.735,Z 413.04,A -85,B 0,C 180,E1 -14181.773,E2 -14181.773} C_VEL
LIN {X 0,Y 340.724,Z 413.041,A -85,B 0,C 180,E1 -14185.595,E2 -14185.595} C_VEL
LIN {X 0,Y 340.699,Z 413.048,A -85,B 0,C 180,E1 -14188.955,E2 -14188.955} C_VEL
LIN {X 0,Y 340.804,Z 413.033,A -85,B 0,C 180,E1 -14193.02,E2 -14193.02} C_VEL
LIN {X 0,Y 340.757,Z 413.036,A -85,B 0,C 180,E1 -14195.638,E2 -14195.638} C_VEL
LIN {X 0,Y 340.754,Z 413.036,A -85,B 0,C 180,E1 -14199.475,E2 -14199.475} C_VEL
LIN {X 0,Y 340.859,Z 413.024,A -85,B 0,C 180,E1 -14201.984,E2 -14201.984} C_VEL
LIN {X 0,Y 340.87,Z 413.022,A -85,B 0,C 180,E1 -14205.705,E2 -14205.705} C_VEL
LIN {X 0,Y 340.877,Z 413.021,A -85,B 0,C 180,E1 -14209.306,E2 -14209.306} C_VEL
LIN {X 0,Y 341.078,Z 412.997,A -85,B 0,C 180,E1 -14212.898,E2 -14212.898} C_VEL
LIN {X 0,Y 341.169,Z 412.985,A -85,B 0,C 180,E1 -14217.639,E2 -14217.639} C_VEL
LIN {X 0,Y 341.318,Z 412.97,A -85,B 0,C 180,E1 -14220,E2 -14220} C_VEL
LIN {X 0,Y 341.169,Z 412.988,A -85,B 0,C 180,E1 -14222.361,E2 -14222.361} C_VEL
LIN {X 0,Y 341.077,Z 412.996,A -85,B 0,C 180,E1 -14227.102,E2 -14227.102} C_VEL
LIN {X 0,Y 340.877,Z 413.021,A -85,B 0,C 180,E1 -14230.694,E2 -14230.694} C_VEL
LIN {X 0,Y 340.864,Z 413.025,A -85,B 0,C 180,E1 -14234.325,E2 -14234.325} C_VEL
LIN {X 0,Y 340.838,Z 413.026,A -85,B 0,C 180,E1 -14238.466,E2 -14238.466} C_VEL
LIN {X 0,Y 340.755,Z 413.041,A -85,B 0,C 180,E1 -14241.857,E2 -14241.857} C_VEL
LIN {X 0,Y 340.773,Z 413.039,A -85,B 0,C 180,E1 -14245.664,E2 -14245.664} C_VEL
LIN {X 0,Y 340.729,Z 413.04,A -85,B 0,C 180,E1 -14248.321,E2 -14248.321} C_VEL
LIN {X 0,Y 340.704,Z 413.043,A -85,B 0,C 180,E1 -14251.044,E2 -14251.044} C_VEL
LIN {X 0,Y 340.72,Z 413.044,A -85,B 0,C 180,E1 -14255.279,E2 -14255.279} C_VEL
LIN {X 0,Y 340.713,Z 413.041,A -85,B 0,C 180,E1 -14258.387,E2 -14258.387} C_VEL
LIN {X 0,Y 340.7,Z 413.044,A -85,B 0,C 180,E1 -14262.046,E2 -14262.046} C_VEL
LIN {X 0,Y 340.686,Z 413.05,A -85,B 0,C 180,E1 -14265.462,E2 -14265.462} C_VEL
LIN {X 0,Y 340.688,Z 413.046,A -85,B 0,C 180,E1 -14268.691,E2 -14268.691} C_VEL
LIN {X 0,Y 340.724,Z 413.044,A -85,B 0,C 180,E1 -14271.772,E2 -14271.772} C_VEL
LIN {X 0,Y 340.633,Z 413.062,A -85,B 0,C 180,E1 -14273.249,E2 -14273.249} C_VEL
LIN {X 0,Y 340.621,Z 415.983,A -85,B 0,C 180,E1 -14276.145,E2 -14276.145} C_VEL
LIN {X 0,Y 340.43,Z 418.912,A -85,B 0,C 180,E1 -14278.928,E2 -14278.928} C_VEL
LIN {X 0,Y 340.2,Z 423.339,A -85,B 0,C 180,E1 -14282.968,E2 -14282.968} C_VEL
LIN {X 0,Y 339.866,Z 427.824,A -85,B 0,C 180,E1 -14286.865,E2 -14286.865} C_VEL
LIN {X 0,Y 339.768,Z 430.011,A -85,B 0,C 180,E1 -14288.685,E2 -14288.685} C_VEL
LIN {X 0,Y 343.314,Z 443.127,A -85,B 0,C 180,E1 -14289.447,E2 -14289.447} C_VEL
LIN {X 0,Y 345.902,Z 454.931,A -85,B 0,C 180,E1 -14290.312,E2 -14290.312} C_VEL
LIN {X 0,Y 347.2,Z 462.457,A -85,B 0,C 180,E1 -14290.955,E2 -14290.955} C_VEL
LIN {X 0,Y 346.166,Z 473.837,A -85,B 0,C 180,E1 -14291.964,E2 -14291.964} C_VEL
LIN {X 0,Y 345.114,Z 484.47,A -85,B 0,C 180,E1 -14293.161,E2 -14293.161} C_VEL
LIN {X 0,Y 343.974,Z 494.721,A -85,B 0,C 180,E1 -14294.597,E2 -14294.597} C_VEL
LIN {X 0,Y 342.749,Z 503.215,A -85,B 0,C 180,E1 -14296.059,E2 -14296.059} C_VEL
LIN {X 0,Y 341.696,Z 511.464,A -85,B 0,C 180,E1 -14297.83,E2 -14297.83} C_VEL
LIN {X 0,Y 340.803,Z 518.109,A -85,B 0,C 180,E1 -14299.605,E2 -14299.605} C_VEL
LIN {X 0,Y 339.993,Z 524.196,A -85,B 0,C 180,E1 -14301.68,E2 -14301.68} C_VEL
LIN {X 0,Y 339.641,Z 527.887,A -85,B 0,C 180,E1 -14303.335,E2 -14303.335} C_VEL
LIN {X 0,Y 339.384,Z 531.06,A -85,B 0,C 180,E1 -14305.249,E2 -14305.249} C_VEL
LIN {X 0,Y 339.192,Z 532.459,A -85,B 0,C 180,E1 -14306.436,E2 -14306.436} C_VEL
LIN {X 0,Y 339.063,Z 534.064,A -85,B 0,C 180,E1 -14308.812,E2 -14308.812} C_VEL
LIN {X 0,Y 339.072,Z 534.295,A -85,B 0,C 180,E1 -14310,E2 -14310} C_VEL
LIN {X 0,Y 339.062,Z 534.105,A -85,B 0,C 180,E1 -14311.188,E2 -14311.188} C_VEL
LIN {X 0,Y 339.187,Z 532.553,A -85,B 0,C 180,E1 -14313.564,E2 -14313.564} C_VEL
LIN {X 0,Y 339.376,Z 531.195,A -85,B 0,C 180,E1 -14314.752,E2 -14314.752} C_VEL
LIN {X 0,Y 339.624,Z 528.141,A -85,B 0,C 180,E1 -14316.64,E2 -14316.64} C_VEL
LIN {X 0,Y 339.991,Z 524.445,A -85,B 0,C 180,E1 -14318.32,E2 -14318.32} C_VEL
LIN {X 0,Y 340.627,Z 519.428,A -85,B 0,C 180,E1 -14320.101,E2 -14320.101} C_VEL
LIN {X 0,Y 341.421,Z 513.113,A -85,B 0,C 180,E1 -14321.879,E2 -14321.879} C_VEL
LIN {X 0,Y 342.514,Z 505.205,A -85,B 0,C 180,E1 -14323.649,E2 -14323.649} C_VEL
LIN {X 0,Y 343.859,Z 495.366,A -85,B 0,C 180,E1 -14325.409,E2 -14325.409} C_VEL
LIN {X 0,Y 344.935,Z 485.486,A -85,B 0,C 180,E1 -14326.821,E2 -14326.821} C_VEL
LIN {X 0,Y 346.093,Z 474.81,A -85,B 0,C 180,E1 -14328.04,E2 -14328.04} C_VEL
LIN {X 0,Y 347.216,Z 462.479,A -85,B 0,C 180,E1 -14329.147,E2 -14329.147} C_VEL
LIN {X 0,Y 345.026,Z 450.794,A -85,B 0,C 180,E1 -14330.122,E2 -14330.122} C_VEL
LIN {X 0,Y 341.992,Z 437.971,A -85,B 0,C 180,E1 -14330.983,E2 -14330.983} C_VEL
LIN {X 0,Y 339.76,Z 429.976,A -85,B 0,C 180,E1 -14331.434,E2 -14331.434} C_VEL
LIN {X 0,Y 339.996,Z 426.271,A -85,B 0,C 180,E1 -14334.561,E2 -14334.561} C_VEL
LIN {X 0,Y 340.209,Z 423.138,A -85,B 0,C 180,E1 -14337.34,E2 -14337.34} C_VEL
LIN {X 0,Y 340.426,Z 419.033,A -85,B 0,C 180,E1 -14341.072,E2 -14341.072} C_VEL
LIN {X 0,Y 340.664,Z 415.558,A -85,B 0,C 180,E1 -14344.39,E2 -14344.39} C_VEL
LIN {X 0,Y 340.66,Z 413.183,A -85,B 0,C 180,E1 -14346.747,E2 -14346.747} C_VEL
LIN {X 0,Y 340.701,Z 413.043,A -85,B 0,C 180,E1 -14349.753,E2 -14349.753} C_VEL
LIN {X 0,Y 340.68,Z 413.05,A -85,B 0,C 180,E1 -14352.904,E2 -14352.904} C_VEL
LIN {X 0,Y 340.668,Z 413.048,A -85,B 0,C 180,E1 -14356.225,E2 -14356.225} C_VEL
LIN {X 0,Y 340.697,Z 413.044,A -85,B 0,C 180,E1 -14358.03,E2 -14358.03} C_VEL
LIN {X 0,Y 340.009,Z 413.134,A -85,B 0,C 180,E1 -14359.017,E2 -14359.017} C_VEL
LIN {X 0,Y 337.167,Z 413.489,A -85,B 0,C 180,E1 -14360.623,E2 -14360.623} C_VEL
LIN {X 0,Y 334.775,Z 413.786,A -85,B 0,C 180,E1 -14361.923,E2 -14361.923} C_VEL
LIN {X 0,Y 333.751,Z 413.912,A -85,B 0,C 180,E1 -14362.929,E2 -14362.929} C_VEL
LIN {X 0,Y 333.668,Z 413.919,A -85,B 0,C 180,E1 -14363.269,E2 -14363.269} C_VEL
LIN {X 0,Y 333.639,Z 413.925,A -85,B 0,C 180,E1 -14366.792,E2 -14366.792} C_VEL
LIN {X 0,Y 333.706,Z 413.914,A -85,B 0,C 180,E1 -14369.71,E2 -14369.71} C_VEL
LIN {X 0,Y 333.742,Z 413.915,A -85,B 0,C 180,E1 -14372.401,E2 -14372.401} C_VEL
LIN {X 0,Y 333.729,Z 413.911,A -85,B 0,C 180,E1 -14375.091,E2 -14375.091} C_VEL
LIN {X 0,Y 333.682,Z 413.917,A -85,B 0,C 180,E1 -14379.019,E2 -14379.019} C_VEL
LIN {X 0,Y 333.796,Z 413.904,A -85,B 0,C 180,E1 -14381.589,E2 -14381.589} C_VEL
LIN {X 0,Y 333.811,Z 413.902,A -85,B 0,C 180,E1 -14385.577,E2 -14385.577} C_VEL
LIN {X 0,Y 333.837,Z 413.898,A -85,B 0,C 180,E1 -14389.078,E2 -14389.078} C_VEL
LIN {X 0,Y 334.029,Z 413.874,A -85,B 0,C 180,E1 -14392.748,E2 -14392.748} C_VEL
LIN {X 0,Y 333.812,Z 413.901,A -85,B 0,C 180,E1 -14395.169,E2 -14395.169} C_VEL
LIN {X 0,Y 334.108,Z 413.867,A -85,B 0,C 180,E1 -14397.589,E2 -14397.589} C_VEL
LIN {X 0,Y 334.249,Z 413.851,A -85,B 0,C 180,E1 -14400,E2 -14400} C_VEL
LIN {X 0,Y 334.108,Z 413.865,A -85,B 0,C 180,E1 -14402.411,E2 -14402.411} C_VEL
LIN {X 0,Y 334.029,Z 413.876,A -85,B 0,C 180,E1 -14407.252,E2 -14407.252} C_VEL
LIN {X 0,Y 333.841,Z 413.898,A -85,B 0,C 180,E1 -14410.922,E2 -14410.922} C_VEL
LIN {X 0,Y 333.811,Z 413.901,A -85,B 0,C 180,E1 -14414.634,E2 -14414.634} C_VEL
LIN {X 0,Y 333.798,Z 413.903,A -85,B 0,C 180,E1 -14418.655,E2 -14418.655} C_VEL
LIN {X 0,Y 333.695,Z 413.915,A -85,B 0,C 180,E1 -14422.278,E2 -14422.278} C_VEL
LIN {X 0,Y 333.737,Z 413.91,A -85,B 0,C 180,E1 -14426.246,E2 -14426.246} C_VEL
LIN {X 0,Y 333.692,Z 413.919,A -85,B 0,C 180,E1 -14428.974,E2 -14428.974} C_VEL
LIN {X 0,Y 333.645,Z 413.921,A -85,B 0,C 180,E1 -14432.587,E2 -14432.587} C_VEL
LIN {X 0,Y 333.679,Z 413.917,A -85,B 0,C 180,E1 -14436.139,E2 -14436.139} C_VEL
LIN {X 0,Y 333.649,Z 413.927,A -85,B 0,C 180,E1 -14439.192,E2 -14439.192} C_VEL
LIN {X 0,Y 333.636,Z 413.927,A -85,B 0,C 180,E1 -14442.5,E2 -14442.5} C_VEL
LIN {X 0,Y 333.681,Z 414.102,A -85,B 0,C 180,E1 -14445.734,E2 -14445.734} C_VEL
LIN {X 0,Y 334.437,Z 418.39,A -85,B 0,C 180,E1 -14449.158,E2 -14449.158} C_VEL
LIN {X 0,Y 334.99,Z 421.872,A -85,B 0,C 180,E1 -14451.764,E2 -14451.764} C_VEL
LIN {X 0,Y 335.265,Z 425.07,A -85,B 0,C 180,E1 -14454.059,E2 -14454.059} C_VEL
LIN {X 0,Y 334.759,Z 429.643,A -85,B 0,C 180,E1 -14457.116,E2 -14457.116} C_VEL
LIN {X 0,Y 334.218,Z 434.653,A -85,B 0,C 180,E1 -14460.385,E2 -14460.385} C_VEL
LIN {X 0,Y 333.527,Z 440.995,A -85,B 0,C 180,E1 -14464.408,E2 -14464.408} C_VEL
LIN {X 0,Y 333.04,Z 447.115,A -85,B 0,C 180,E1 -14468.145,E2 -14468.145} C_VEL
LIN {X 0,Y 335.987,Z 460.576,A -85,B 0,C 180,E1 -14468.872,E2 -14468.872} C_VEL
LIN {X 0,Y 338.066,Z 473.382,A -85,B 0,C 180,E1 -14469.772,E2 -14469.772} C_VEL
LIN {X 0,Y 339.261,Z 485.268,A -85,B 0,C 180,E1 -14470.8,E2 -14470.8} C_VEL
LIN {X 0,Y 338.938,Z 491.66,A -85,B 0,C 180,E1 -14471.409,E2 -14471.409} C_VEL
LIN {X 0,Y 337.462,Z 503.448,A -85,B 0,C 180,E1 -14472.736,E2 -14472.736} C_VEL
LIN {X 0,Y 336.243,Z 513.923,A -85,B 0,C 180,E1 -14474.233,E2 -14474.233} C_VEL
LIN {X 0,Y 335.142,Z 522.402,A -85,B 0,C 180,E1 -14475.735,E2 -14475.735} C_VEL
LIN {X 0,Y 333.914,Z 530.674,A -85,B 0,C 180,E1 -14477.541,E2 -14477.541} C_VEL
LIN {X 0,Y 333.118,Z 537.348,A -85,B 0,C 180,E1 -14479.362,E2 -14479.362} C_VEL
LIN {X 0,Y 332.479,Z 543.457,A -85,B 0,C 180,E1 -14481.491,E2 -14481.491} C_VEL
LIN {X 0,Y 332.108,Z 547.427,A -85,B 0,C 180,E1 -14483.316,E2 -14483.316} C_VEL
LIN {X 0,Y 331.981,Z 550.363,A -85,B 0,C 180,E1 -14485.142,E2 -14485.142} C_VEL
LIN {X 0,Y 331.997,Z 551.762,A -85,B 0,C 180,E1 -14486.359,E2 -14486.359} C_VEL
LIN {X 0,Y 331.924,Z 553.366,A -85,B 0,C 180,E1 -14488.787,E2 -14488.787} C_VEL
LIN {X 0,Y 331.97,Z 553.582,A -85,B 0,C 180,E1 -14490,E2 -14490} C_VEL
LIN {X 0,Y 331.924,Z 553.361,A -85,B 0,C 180,E1 -14491.213,E2 -14491.213} C_VEL
LIN {X 0,Y 331.997,Z 551.752,A -85,B 0,C 180,E1 -14493.641,E2 -14493.641} C_VEL
LIN {X 0,Y 332.009,Z 548.974,A -85,B 0,C 180,E1 -14495.787,E2 -14495.787} C_VEL
LIN {X 0,Y 332.359,Z 544.857,A -85,B 0,C 180,E1 -14497.9,E2 -14497.9} C_VEL
LIN {X 0,Y 332.8,Z 540.124,A -85,B 0,C 180,E1 -14499.726,E2 -14499.726} C_VEL
LIN {X 0,Y 333.585,Z 533.017,A -85,B 0,C 180,E1 -14501.854,E2 -14501.854} C_VEL
LIN {X 0,Y 334.717,Z 525.311,A -85,B 0,C 180,E1 -14503.663,E2 -14503.663} C_VEL
LIN {X 0,Y 335.761,Z 517.421,A -85,B 0,C 180,E1 -14505.168,E2 -14505.168} C_VEL
LIN {X 0,Y 336.918,Z 507.711,A -85,B 0,C 180,E1 -14506.68,E2 -14506.68} C_VEL
LIN {X 0,Y 338.256,Z 497.119,A -85,B 0,C 180,E1 -14508.003,E2 -14508.003} C_VEL
LIN {X 0,Y 339.312,Z 486.796,A -85,B 0,C 180,E1 -14509.04,E2 -14509.04} C_VEL
LIN {X 0,Y 338.233,Z 474.588,A -85,B 0,C 180,E1 -14510.117,E2 -14510.117} C_VEL
LIN {X 0,Y 336.113,Z 461.223,A -85,B 0,C 180,E1 -14511.068,E2 -14511.068} C_VEL
LIN {X 0,Y 333.238,Z 448.391,A -85,B 0,C 180,E1 -14511.787,E2 -14511.787} C_VEL
LIN {X 0,Y 333.04,Z 446.885,A -85,B 0,C 180,E1 -14511.874,E2 -14511.874} C_VEL
LIN {X 0,Y 333.522,Z 440.964,A -85,B 0,C 180,E1 -14515.592,E2 -14515.592} C_VEL
LIN {X 0,Y 334.249,Z 434.61,A -85,B 0,C 180,E1 -14519.611,E2 -14519.611} C_VEL
LIN {X 0,Y 334.802,Z 429.304,A -85,B 0,C 180,E1 -14523.078,E2 -14523.078} C_VEL
LIN {X 0,Y 335.198,Z 425.031,A -85,B 0,C 180,E1 -14525.949,E2 -14525.949} C_VEL
LIN {X 0,Y 334.853,Z 420.716,A -85,B 0,C 180,E1 -14529.053,E2 -14529.053} C_VEL
LIN {X 0,Y 334.096,Z 416.139,A -85,B 0,C 180,E1 -14532.586,E2 -14532.586} C_VEL
LIN {X 0,Y 333.661,Z 413.926,A -85,B 0,C 180,E1 -14534.464,E2 -14534.464} C_VEL
LIN {X 0,Y 333.642,Z 413.924,A -85,B 0,C 180,E1 -14537.618,E2 -14537.618} C_VEL
LIN {X 0,Y 333.654,Z 413.926,A -85,B 0,C 180,E1 -14541.202,E2 -14541.202} C_VEL
LIN {X 0,Y 333.677,Z 413.919,A -85,B 0,C 180,E1 -14543.861,E2 -14543.861} C_VEL
LIN {X 0,Y 333.644,Z 413.924,A -85,B 0,C 180,E1 -14547.413,E2 -14547.413} C_VEL
LIN {X 0,Y 333.691,Z 413.92,A -85,B 0,C 180,E1 -14551.026,E2 -14551.026} C_VEL
LIN {X 0,Y 333.736,Z 413.91,A -85,B 0,C 180,E1 -14553.754,E2 -14553.754} C_VEL
LIN {X 0,Y 333.72,Z 413.913,A -85,B 0,C 180,E1 -14557.914,E2 -14557.914} C_VEL
LIN {X 0,Y 333.795,Z 413.903,A -85,B 0,C 180,E1 -14561.589,E2 -14561.589} C_VEL
LIN {X 0,Y 333.809,Z 413.901,A -85,B 0,C 180,E1 -14565.577,E2 -14565.577} C_VEL
LIN {X 0,Y 333.839,Z 413.898,A -85,B 0,C 180,E1 -14569.078,E2 -14569.078} C_VEL
LIN {X 0,Y 334.027,Z 413.876,A -85,B 0,C 180,E1 -14572.748,E2 -14572.748} C_VEL
LIN {X 0,Y 333.811,Z 413.901,A -85,B 0,C 180,E1 -14575.169,E2 -14575.169} C_VEL
LIN {X 0,Y 334.107,Z 413.865,A -85,B 0,C 180,E1 -14577.589,E2 -14577.589} C_VEL
LIN {X 0,Y 334.268,Z 413.848,A -85,B 0,C 180,E1 -14580,E2 -14580} C_VEL
LIN {X 0,Y 334.107,Z 413.868,A -85,B 0,C 180,E1 -14582.411,E2 -14582.411} C_VEL
LIN {X 0,Y 334.027,Z 413.874,A -85,B 0,C 180,E1 -14587.253,E2 -14587.253} C_VEL
LIN {X 0,Y 333.839,Z 413.897,A -85,B 0,C 180,E1 -14590.922,E2 -14590.922} C_VEL
LIN {X 0,Y 333.81,Z 413.902,A -85,B 0,C 180,E1 -14594.634,E2 -14594.634} C_VEL
LIN {X 0,Y 333.797,Z 413.902,A -85,B 0,C 180,E1 -14598.655,E2 -14598.655} C_VEL
LIN {X 0,Y 333.694,Z 413.917,A -85,B 0,C 180,E1 -14602.278,E2 -14602.278} C_VEL
LIN {X 0,Y 333.736,Z 413.912,A -85,B 0,C 180,E1 -14606.246,E2 -14606.246} C_VEL
LIN {X 0,Y 333.705,Z 413.915,A -85,B 0,C 180,E1 -14610.29,E2 -14610.29} C_VEL
LIN {X 0,Y 333.676,Z 413.918,A -85,B 0,C 180,E1 -14614.659,E2 -14614.659} C_VEL
LIN {X 0,Y 333.656,Z 413.925,A -85,B 0,C 180,E1 -14617.651,E2 -14617.651} C_VEL
LIN {X 0,Y 333.648,Z 413.922,A -85,B 0,C 180,E1 -14620.768,E2 -14620.768} C_VEL
LIN {X 0,Y 333.626,Z 413.925,A -85,B 0,C 180,E1 -14624.256,E2 -14624.256} C_VEL
LIN {X 0,Y 333.644,Z 413.925,A -85,B 0,C 180,E1 -14627.619,E2 -14627.619} C_VEL
LIN {X 0,Y 333.648,Z 413.927,A -85,B 0,C 180,E1 -14631.203,E2 -14631.203} C_VEL
LIN {X 0,Y 333.603,Z 414.033,A -85,B 0,C 180,E1 -14633.183,E2 -14633.183} C_VEL
LIN {X 0,Y 333.636,Z 416.158,A -85,B 0,C 180,E1 -14635.337,E2 -14635.337} C_VEL
LIN {X 0,Y 333.433,Z 419.088,A -85,B 0,C 180,E1 -14638.201,E2 -14638.201} C_VEL
LIN {X 0,Y 333.251,Z 422.045,A -85,B 0,C 180,E1 -14640.984,E2 -14640.984} C_VEL
LIN {X 0,Y 333.056,Z 425.018,A -85,B 0,C 180,E1 -14643.696,E2 -14643.696} C_VEL
LIN {X 0,Y 332.737,Z 429.539,A -85,B 0,C 180,E1 -14647.654,E2 -14647.654} C_VEL
LIN {X 0,Y 332.729,Z 430.277,A -85,B 0,C 180,E1 -14648.212,E2 -14648.212} C_VEL
LIN {X 0,Y 336.391,Z 443.463,A -85,B 0,C 180,E1 -14649.01,E2 -14649.01} C_VEL
LIN {X 0,Y 339.076,Z 455.694,A -85,B 0,C 180,E1 -14649.938,E2 -14649.938} C_VEL
LIN {X 0,Y 340.403,Z 464.375,A -85,B 0,C 180,E1 -14650.711,E2 -14650.711} C_VEL
LIN {X 0,Y 339.272,Z 475.467,A -85,B 0,C 180,E1 -14651.741,E2 -14651.741} C_VEL
LIN {X 0,Y 338.266,Z 485.255,A -85,B 0,C 180,E1 -14652.887,E2 -14652.887} C_VEL
LIN {X 0,Y 337.131,Z 494.928,A -85,B 0,C 180,E1 -14654.276,E2 -14654.276} C_VEL
LIN {X 0,Y 335.871,Z 503.422,A -85,B 0,C 180,E1 -14655.767,E2 -14655.767} C_VEL
LIN {X 0,Y 334.773,Z 511.67,A -85,B 0,C 180,E1 -14657.574,E2 -14657.574} C_VEL
LIN {X 0,Y 333.834,Z 518.314,A -85,B 0,C 180,E1 -14659.385,E2 -14659.385} C_VEL
LIN {X 0,Y 332.948,Z 524.402,A -85,B 0,C 180,E1 -14661.503,E2 -14661.503} C_VEL
LIN {X 0,Y 332.557,Z 528.39,A -85,B 0,C 180,E1 -14663.348,E2 -14663.348} C_VEL
LIN {X 0,Y 332.306,Z 531.265,A -85,B 0,C 180,E1 -14665.147,E2 -14665.147} C_VEL
LIN {X 0,Y 332.123,Z 532.663,A -85,B 0,C 180,E1 -14666.36,E2 -14666.36} C_VEL
LIN {X 0,Y 331.968,Z 534.268,A -85,B 0,C 180,E1 -14668.787,E2 -14668.787} C_VEL
LIN {X 0,Y 331.975,Z 534.499,A -85,B 0,C 180,E1 -14670,E2 -14670} C_VEL
LIN {X 0,Y 331.968,Z 534.309,A -85,B 0,C 180,E1 -14671.213,E2 -14671.213} C_VEL
LIN {X 0,Y 332.118,Z 532.756,A -85,B 0,C 180,E1 -14673.64,E2 -14673.64} C_VEL
LIN {X 0,Y 332.298,Z 531.398,A -85,B 0,C 180,E1 -14674.853,E2 -14674.853} C_VEL
LIN {X 0,Y 332.543,Z 528.608,A -85,B 0,C 180,E1 -14676.632,E2 -14676.632} C_VEL
LIN {X 0,Y 332.944,Z 524.648,A -85,B 0,C 180,E1 -14678.497,E2 -14678.497} C_VEL
LIN {X 0,Y 333.632,Z 519.631,A -85,B 0,C 180,E1 -14680.315,E2 -14680.315} C_VEL
LIN {X 0,Y 334.48,Z 513.315,A -85,B 0,C 180,E1 -14682.129,E2 -14682.129} C_VEL
LIN {X 0,Y 335.596,Z 505.407,A -85,B 0,C 180,E1 -14683.936,E2 -14683.936} C_VEL
LIN {X 0,Y 337.015,Z 495.567,A -85,B 0,C 180,E1 -14685.73,E2 -14685.73} C_VEL
LIN {X 0,Y 338.146,Z 485.686,A -85,B 0,C 180,E1 -14687.169,E2 -14687.169} C_VEL
LIN {X 0,Y 339.354,Z 475.009,A -85,B 0,C 180,E1 -14688.411,E2 -14688.411} C_VEL
LIN {X 0,Y 340.453,Z 463.793,A -85,B 0,C 180,E1 -14689.445,E2 -14689.445} C_VEL
LIN {X 0,Y 338.4,Z 452.398,A -85,B 0,C 180,E1 -14690.445,E2 -14690.445} C_VEL
LIN {X 0,Y 335.405,Z 439.652,A -85,B 0,C 180,E1 -14691.35,E2 -14691.35} C_VEL
LIN {X 0,Y 332.728,Z 430.152,A -85,B 0,C 180,E1 -14691.93,E2 -14691.93} C_VEL
LIN {X 0,Y 332.949,Z 426.629,A -85,B 0,C 180,E1 -14694.972,E2 -14694.972} C_VEL
LIN {X 0,Y 333.175,Z 423.663,A -85,B 0,C 180,E1 -14697.65,E2 -14697.65} C_VEL
LIN {X 0,Y 333.346,Z 420.693,A -85,B 0,C 180,E1 -14700.398,E2 -14700.398} C_VEL
LIN {X 0,Y 333.549,Z 417.747,A -85,B 0,C 180,E1 -14703.218,E2 -14703.218} C_VEL
LIN {X 0,Y 333.656,Z 414.805,A -85,B 0,C 180,E1 -14706.142,E2 -14706.142} C_VEL
LIN {X 0,Y 333.627,Z 414.142,A -85,B 0,C 180,E1 -14706.823,E2 -14706.823} C_VEL
LIN {X 0,Y 333.646,Z 413.924,A -85,B 0,C 180,E1 -14709.193,E2 -14709.193} C_VEL
LIN {X 0,Y 333.636,Z 413.926,A -85,B 0,C 180,E1 -14712.5,E2 -14712.5} C_VEL
LIN {X 0,Y 333.622,Z 413.925,A -85,B 0,C 180,E1 -14715.959,E2 -14715.959} C_VEL
LIN {X 0,Y 333.649,Z 413.922,A -85,B 0,C 180,E1 -14719.315,E2 -14719.315} C_VEL
LIN {X 0,Y 333.668,Z 413.919,A -85,B 0,C 180,E1 -14723.269,E2 -14723.269} C_VEL
LIN {X 0,Y 332.991,Z 414.007,A -85,B 0,C 180,E1 -14724.277,E2 -14724.277} C_VEL
LIN {X 0,Y 330.104,Z 414.364,A -85,B 0,C 180,E1 -14725.915,E2 -14725.915} C_VEL
LIN {X 0,Y 327.674,Z 414.665,A -85,B 0,C 180,E1 -14727.243,E2 -14727.243} C_VEL
LIN {X 0,Y 326.654,Z 414.796,A -85,B 0,C 180,E1 -14728.271,E2 -14728.271} C_VEL
LIN {X 0,Y 326.583,Z 414.801,A -85,B 0,C 180,E1 -14728.619,E2 -14728.619} C_VEL
LIN {X 0,Y 326.661,Z 414.793,A -85,B 0,C 180,E1 -14731.897,E2 -14731.897} C_VEL
LIN {X 0,Y 326.691,Z 414.791,A -85,B 0,C 180,E1 -14734.627,E2 -14734.627} C_VEL
LIN {X 0,Y 326.648,Z 414.796,A -85,B 0,C 180,E1 -14738.545,E2 -14738.545} C_VEL
LIN {X 0,Y 326.747,Z 414.781,A -85,B 0,C 180,E1 -14741.178,E2 -14741.178} C_VEL
LIN {X 0,Y 326.766,Z 414.779,A -85,B 0,C 180,E1 -14745.433,E2 -14745.433} C_VEL
LIN {X 0,Y 326.773,Z 414.778,A -85,B 0,C 180,E1 -14748.839,E2 -14748.839} C_VEL
LIN {X 0,Y 326.982,Z 414.753,A -85,B 0,C 180,E1 -14752.59,E2 -14752.59} C_VEL
LIN {X 0,Y 326.779,Z 414.777,A -85,B 0,C 180,E1 -14755.065,E2 -14755.065} C_VEL
LIN {X 0,Y 327.048,Z 414.746,A -85,B 0,C 180,E1 -14757.537,E2 -14757.537} C_VEL
LIN {X 0,Y 327.2,Z 414.729,A -85,B 0,C 180,E1 -14760,E2 -14760} C_VEL
LIN {X 0,Y 327.049,Z 414.744,A -85,B 0,C 180,E1 -14762.463,E2 -14762.463} C_VEL
LIN {X 0,Y 326.999,Z 414.751,A -85,B 0,C 180,E1 -14766.169,E2 -14766.169} C_VEL
LIN {X 0,Y 326.917,Z 414.76,A -85,B 0,C 180,E1 -14768.655,E2 -14768.655} C_VEL
LIN {X 0,Y 326.741,Z 414.782,A -85,B 0,C 180,E1 -14772.421,E2 -14772.421} C_VEL
LIN {X 0,Y 326.757,Z 414.781,A -85,B 0,C 180,E1 -14774.957,E2 -14774.957} C_VEL
LIN {X 0,Y 326.735,Z 414.783,A -85,B 0,C 180,E1 -14778.838,E2 -14778.838} C_VEL
LIN {X 0,Y 326.623,Z 414.797,A -85,B 0,C 180,E1 -14782.787,E2 -14782.787} C_VEL
LIN {X 0,Y 326.692,Z 414.792,A -85,B 0,C 180,E1 -14785.484,E2 -14785.484} C_VEL
LIN {X 0,Y 326.65,Z 414.795,A -85,B 0,C 180,E1 -14789.66,E2 -14789.66} C_VEL
LIN {X 0,Y 326.609,Z 414.798,A -85,B 0,C 180,E1 -14794.019,E2 -14794.019} C_VEL
LIN {X 0,Y 326.63,Z 414.8,A -85,B 0,C 180,E1 -14797.239,E2 -14797.239} C_VEL
LIN {X 0,Y 326.58,Z 414.808,A -85,B 0,C 180,E1 -14801.131,E2 -14801.131} C_VEL
LIN {X 0,Y 326.613,Z 414.798,A -85,B 0,C 180,E1 -14805.168,E2 -14805.168} C_VEL
LIN {X 0,Y 327.357,Z 419.065,A -85,B 0,C 180,E1 -14808.713,E2 -14808.713} C_VEL
LIN {X 0,Y 327.956,Z 422.755,A -85,B 0,C 180,E1 -14811.577,E2 -14811.577} C_VEL
LIN {X 0,Y 328.198,Z 427.053,A -85,B 0,C 180,E1 -14814.677,E2 -14814.677} C_VEL
LIN {X 0,Y 327.554,Z 432.363,A -85,B 0,C 180,E1 -14818.286,E2 -14818.286} C_VEL
LIN {X 0,Y 326.894,Z 437.714,A -85,B 0,C 180,E1 -14821.821,E2 -14821.821} C_VEL
LIN {X 0,Y 326.227,Z 443.93,A -85,B 0,C 180,E1 -14825.838,E2 -14825.838} C_VEL
LIN {X 0,Y 326.034,Z 446.77,A -85,B 0,C 180,E1 -14827.646,E2 -14827.646} C_VEL
LIN {X 0,Y 328.964,Z 460.015,A -85,B 0,C 180,E1 -14828.38,E2 -14828.38} C_VEL
LIN {X 0,Y 331.182,Z 473.178,A -85,B 0,C 180,E1 -14829.332,E2 -14829.332} C_VEL
LIN {X 0,Y 332.362,Z 485.063,A -85,B 0,C 180,E1 -14830.386,E2 -14830.386} C_VEL
LIN {X 0,Y 332.379,Z 489.928,A -85,B 0,C 180,E1 -14830.868,E2 -14830.868} C_VEL
LIN {X 0,Y 331.003,Z 500.893,A -85,B 0,C 180,E1 -14832.069,E2 -14832.069} C_VEL
LIN {X 0,Y 329.661,Z 511.235,A -85,B 0,C 180,E1 -14833.504,E2 -14833.504} C_VEL
LIN {X 0,Y 328.393,Z 520.614,A -85,B 0,C 180,E1 -14835.119,E2 -14835.119} C_VEL
LIN {X 0,Y 327.362,Z 527.915,A -85,B 0,C 180,E1 -14836.656,E2 -14836.656} C_VEL
LIN {X 0,Y 326.347,Z 535.106,A -85,B 0,C 180,E1 -14838.51,E2 -14838.51} C_VEL
LIN {X 0,Y 325.593,Z 541.66,A -85,B 0,C 180,E1 -14840.683,E2 -14840.683} C_VEL
LIN {X 0,Y 325.157,Z 545.998,A -85,B 0,C 180,E1 -14842.548,E2 -14842.548} C_VEL
LIN {X 0,Y 324.914,Z 549.054,A -85,B 0,C 180,E1 -14844.267,E2 -14844.267} C_VEL
LIN {X 0,Y 324.901,Z 551.558,A -85,B 0,C 180,E1 -14846.279,E2 -14846.279} C_VEL
LIN {X 0,Y 324.832,Z 553.162,A -85,B 0,C 180,E1 -14848.76,E2 -14848.76} C_VEL
LIN {X 0,Y 324.875,Z 553.378,A -85,B 0,C 180,E1 -14850,E2 -14850} C_VEL
LIN {X 0,Y 324.832,Z 553.157,A -85,B 0,C 180,E1 -14851.24,E2 -14851.24} C_VEL
LIN {X 0,Y 324.9,Z 551.547,A -85,B 0,C 180,E1 -14853.721,E2 -14853.721} C_VEL
LIN {X 0,Y 324.914,Z 549.035,A -85,B 0,C 180,E1 -14855.733,E2 -14855.733} C_VEL
LIN {X 0,Y 325.157,Z 545.967,A -85,B 0,C 180,E1 -14857.451,E2 -14857.451} C_VEL
LIN {X 0,Y 325.593,Z 541.618,A -85,B 0,C 180,E1 -14859.316,E2 -14859.316} C_VEL
LIN {X 0,Y 326.224,Z 536.08,A -85,B 0,C 180,E1 -14861.18,E2 -14861.18} C_VEL
LIN {X 0,Y 327.188,Z 529.172,A -85,B 0,C 180,E1 -14863.035,E2 -14863.035} C_VEL
LIN {X 0,Y 328.208,Z 522.121,A -85,B 0,C 180,E1 -14864.572,E2 -14864.572} C_VEL
LIN {X 0,Y 329.387,Z 513.623,A -85,B 0,C 180,E1 -14866.104,E2 -14866.104} C_VEL
LIN {X 0,Y 330.656,Z 503.121,A -85,B 0,C 180,E1 -14867.631,E2 -14867.631} C_VEL
LIN {X 0,Y 332.196,Z 491.308,A -85,B 0,C 180,E1 -14868.982,E2 -14868.982} C_VEL
LIN {X 0,Y 332.416,Z 486.581,A -85,B 0,C 180,E1 -14869.45,E2 -14869.45} C_VEL
LIN {X 0,Y 331.303,Z 474.369,A -85,B 0,C 180,E1 -14870.556,E2 -14870.556} C_VEL
LIN {X 0,Y 329.205,Z 461.303,A -85,B 0,C 180,E1 -14871.515,E2 -14871.515} C_VEL
LIN {X 0,Y 326.386,Z 448.728,A -85,B 0,C 180,E1 -14872.25,E2 -14872.25} C_VEL
LIN {X 0,Y 326.011,Z 446.719,A -85,B 0,C 180,E1 -14872.354,E2 -14872.354} C_VEL
LIN {X 0,Y 326.542,Z 440.768,A -85,B 0,C 180,E1 -14876.181,E2 -14876.181} C_VEL
LIN {X 0,Y 327.203,Z 435.49,A -85,B 0,C 180,E1 -14879.605,E2 -14879.605} C_VEL
LIN {X 0,Y 327.804,Z 430.02,A -85,B 0,C 180,E1 -14883.264,E2 -14883.264} C_VEL
LIN {X 0,Y 328.168,Z 426.704,A -85,B 0,C 180,E1 -14885.531,E2 -14885.531} C_VEL
LIN {X 0,Y 327.971,Z 422.719,A -85,B 0,C 180,E1 -14888.421,E2 -14888.421} C_VEL
LIN {X 0,Y 327.275,Z 418.472,A -85,B 0,C 180,E1 -14891.736,E2 -14891.736} C_VEL
LIN {X 0,Y 326.566,Z 414.811,A -85,B 0,C 180,E1 -14894.901,E2 -14894.901} C_VEL
LIN {X 0,Y 326.579,Z 414.807,A -85,B 0,C 180,E1 -14898.869,E2 -14898.869} C_VEL
LIN {X 0,Y 326.629,Z 414.801,A -85,B 0,C 180,E1 -14902.761,E2 -14902.761} C_VEL
LIN {X 0,Y 326.608,Z 414.8,A -85,B 0,C 180,E1 -14905.981,E2 -14905.981} C_VEL
LIN {X 0,Y 326.649,Z 414.796,A -85,B 0,C 180,E1 -14910.34,E2 -14910.34} C_VEL
LIN {X 0,Y 326.691,Z 414.792,A -85,B 0,C 180,E1 -14914.516,E2 -14914.516} C_VEL
LIN {X 0,Y 326.649,Z 414.798,A -85,B 0,C 180,E1 -14918.545,E2 -14918.545} C_VEL
LIN {X 0,Y 326.745,Z 414.783,A -85,B 0,C 180,E1 -14921.178,E2 -14921.178} C_VEL
LIN {X 0,Y 326.764,Z 414.779,A -85,B 0,C 180,E1 -14925.433,E2 -14925.433} C_VEL
LIN {X 0,Y 326.775,Z 414.78,A -85,B 0,C 180,E1 -14928.839,E2 -14928.839} C_VEL
LIN {X 0,Y 326.981,Z 414.755,A -85,B 0,C 180,E1 -14932.59,E2 -14932.59} C_VEL
LIN {X 0,Y 326.778,Z 414.777,A -85,B 0,C 180,E1 -14935.065,E2 -14935.065} C_VEL
LIN {X 0,Y 327.047,Z 414.744,A -85,B 0,C 180,E1 -14937.537,E2 -14937.537} C_VEL
LIN {X 0,Y 327.219,Z 414.726,A -85,B 0,C 180,E1 -14940,E2 -14940} C_VEL
LIN {X 0,Y 327.047,Z 414.746,A -85,B 0,C 180,E1 -14942.463,E2 -14942.463} C_VEL
LIN {X 0,Y 326.973,Z 414.754,A -85,B 0,C 180,E1 -14946.674,E2 -14946.674} C_VEL
LIN {X 0,Y 326.817,Z 414.777,A -85,B 0,C 180,E1 -14949.906,E2 -14949.906} C_VEL
LIN {X 0,Y 326.762,Z 414.782,A -85,B 0,C 180,E1 -14953.685,E2 -14953.685} C_VEL
LIN {X 0,Y 326.701,Z 414.789,A -85,B 0,C 180,E1 -14957.528,E2 -14957.528} C_VEL
LIN {X 0,Y 326.664,Z 414.794,A -85,B 0,C 180,E1 -14960.135,E2 -14960.135} C_VEL
LIN {X 0,Y 326.653,Z 414.795,A -85,B 0,C 180,E1 -14964.129,E2 -14964.129} C_VEL
LIN {X 0,Y 326.684,Z 414.789,A -85,B 0,C 180,E1 -14966.858,E2 -14966.858} C_VEL
LIN {X 0,Y 326.641,Z 414.794,A -85,B 0,C 180,E1 -14970.612,E2 -14970.612} C_VEL
LIN {X 0,Y 326.609,Z 414.8,A -85,B 0,C 180,E1 -14974.019,E2 -14974.019} C_VEL
LIN {X 0,Y 326.631,Z 414.799,A -85,B 0,C 180,E1 -14977.239,E2 -14977.239} C_VEL
LIN {X 0,Y 326.579,Z 414.805,A -85,B 0,C 180,E1 -14981.132,E2 -14981.132} C_VEL
LIN {X 0,Y 326.557,Z 414.806,A -85,B 0,C 180,E1 -14984.748,E2 -14984.748} C_VEL
LIN {X 0,Y 326.578,Z 414.803,A -85,B 0,C 180,E1 -14988.155,E2 -14988.155} C_VEL
LIN {X 0,Y 326.591,Z 414.806,A -85,B 0,C 180,E1 -14991.387,E2 -14991.387} C_VEL
LIN {X 0,Y 326.582,Z 414.859,A -85,B 0,C 180,E1 -14992.947,E2 -14992.947} C_VEL
LIN {X 0,Y 326.553,Z 417.79,A -85,B 0,C 180,E1 -14995.974,E2 -14995.974} C_VEL
LIN {X 0,Y 326.316,Z 421.379,A -85,B 0,C 180,E1 -14999.486,E2 -14999.486} C_VEL
LIN {X 0,Y 326.041,Z 425.21,A -85,B 0,C 180,E1 -15003.085,E2 -15003.085} C_VEL
LIN {X 0,Y 325.813,Z 428.223,A -85,B 0,C 180,E1 -15005.805,E2 -15005.805} C_VEL
LIN {X 0,Y 325.689,Z 430.513,A -85,B 0,C 180,E1 -15007.716,E2 -15007.716} C_VEL
LIN {X 0,Y 329.435,Z 443.799,A -85,B 0,C 180,E1 -15008.551,E2 -15008.551} C_VEL
LIN {X 0,Y 332.269,Z 456.495,A -85,B 0,C 180,E1 -15009.55,E2 -15009.55} C_VEL
LIN {X 0,Y 333.574,Z 464.589,A -85,B 0,C 180,E1 -15010.3,E2 -15010.3} C_VEL
LIN {X 0,Y 332.734,Z 474.254,A -85,B 0,C 180,E1 -15011.21,E2 -15011.21} C_VEL
LIN {X 0,Y 331.52,Z 484.887,A -85,B 0,C 180,E1 -15012.449,E2 -15012.449} C_VEL
LIN {X 0,Y 330.31,Z 495.135,A -85,B 0,C 180,E1 -15013.943,E2 -15013.943} C_VEL
LIN {X 0,Y 329.001,Z 503.628,A -85,B 0,C 180,E1 -15015.463,E2 -15015.463} C_VEL
LIN {X 0,Y 327.851,Z 511.876,A -85,B 0,C 180,E1 -15017.307,E2 -15017.307} C_VEL
LIN {X 0,Y 326.97,Z 517.52,A -85,B 0,C 180,E1 -15018.846,E2 -15018.846} C_VEL
LIN {X 0,Y 326.124,Z 523.02,A -85,B 0,C 180,E1 -15020.699,E2 -15020.699} C_VEL
LIN {X 0,Y 325.622,Z 527.333,A -85,B 0,C 180,E1 -15022.559,E2 -15022.559} C_VEL
LIN {X 0,Y 325.393,Z 529.615,A -85,B 0,C 180,E1 -15023.801,E2 -15023.801} C_VEL
LIN {X 0,Y 325.231,Z 531.47,A -85,B 0,C 180,E1 -15025.041,E2 -15025.041} C_VEL
LIN {X 0,Y 325.056,Z 532.867,A -85,B 0,C 180,E1 -15026.281,E2 -15026.281} C_VEL
LIN {X 0,Y 324.876,Z 534.472,A -85,B 0,C 180,E1 -15028.761,E2 -15028.761} C_VEL
LIN {X 0,Y 324.88,Z 534.703,A -85,B 0,C 180,E1 -15030,E2 -15030} C_VEL
LIN {X 0,Y 324.876,Z 534.512,A -85,B 0,C 180,E1 -15031.24,E2 -15031.24} C_VEL
LIN {X 0,Y 325.052,Z 532.959,A -85,B 0,C 180,E1 -15033.719,E2 -15033.719} C_VEL
LIN {X 0,Y 325.223,Z 531.602,A -85,B 0,C 180,E1 -15034.959,E2 -15034.959} C_VEL
LIN {X 0,Y 325.45,Z 529.103,A -85,B 0,C 180,E1 -15036.605,E2 -15036.605} C_VEL
LIN {X 0,Y 325.907,Z 524.851,A -85,B 0,C 180,E1 -15038.682,E2 -15038.682} C_VEL
LIN {X 0,Y 326.647,Z 519.834,A -85,B 0,C 180,E1 -15040.538,E2 -15040.538} C_VEL
LIN {X 0,Y 327.546,Z 513.517,A -85,B 0,C 180,E1 -15042.39,E2 -15042.39} C_VEL
LIN {X 0,Y 328.702,Z 505.609,A -85,B 0,C 180,E1 -15044.234,E2 -15044.234} C_VEL
LIN {X 0,Y 330.188,Z 495.768,A -85,B 0,C 180,E1 -15046.064,E2 -15046.064} C_VEL
LIN {X 0,Y 331.417,Z 485.441,A -85,B 0,C 180,E1 -15047.589,E2 -15047.589} C_VEL
LIN {X 0,Y 332.638,Z 475.208,A -85,B 0,C 180,E1 -15048.796,E2 -15048.796} C_VEL
LIN {X 0,Y 333.631,Z 465.768,A -85,B 0,C 180,E1 -15049.697,E2 -15049.697} C_VEL
LIN {X 0,Y 332.016,Z 455.513,A -85,B 0,C 180,E1 -15050.646,E2 -15050.646} C_VEL
LIN {X 0,Y 329.203,Z 442.777,A -85,B 0,C 180,E1 -15051.63,E2 -15051.63} C_VEL
LIN {X 0,Y 325.694,Z 430.379,A -85,B 0,C 180,E1 -15052.404,E2 -15052.404} C_VEL
LIN {X 0,Y 325.936,Z 426.825,A -85,B 0,C 180,E1 -15055.547,E2 -15055.547} C_VEL
LIN {X 0,Y 326.15,Z 423.851,A -85,B 0,C 180,E1 -15058.299,E2 -15058.299} C_VEL
LIN {X 0,Y 326.34,Z 420.877,A -85,B 0,C 180,E1 -15061.122,E2 -15061.122} C_VEL
LIN {X 0,Y 326.563,Z 417.91,A -85,B 0,C 180,E1 -15064.025,E2 -15064.025} C_VEL
LIN {X 0,Y 326.568,Z 414.814,A -85,B 0,C 180,E1 -15067.224,E2 -15067.224} C_VEL
LIN {X 0,Y 326.593,Z 414.801,A -85,B 0,C 180,E1 -15070.209,E2 -15070.209} C_VEL
LIN {X 0,Y 326.58,Z 414.802,A -85,B 0,C 180,E1 -15073.523,E2 -15073.523} C_VEL
LIN {X 0,Y 326.584,Z 414.804,A -85,B 0,C 180,E1 -15077.027,E2 -15077.027} C_VEL
LIN {X 0,Y 326.614,Z 414.802,A -85,B 0,C 180,E1 -15080.773,E2 -15080.773} C_VEL
LIN {X 0,Y 326.616,Z 414.802,A -85,B 0,C 180,E1 -15084.481,E2 -15084.481} C_VEL
LIN {X 0,Y 326.61,Z 414.798,A -85,B 0,C 180,E1 -15087.456,E2 -15087.456} C_VEL
LIN {X 0,Y 326.583,Z 414.801,A -85,B 0,C 180,E1 -15088.619,E2 -15088.619} C_VEL
LIN {X 0,Y 325.955,Z 414.883,A -85,B 0,C 180,E1 -15089.649,E2 -15089.649} C_VEL
LIN {X 0,Y 323.144,Z 415.233,A -85,B 0,C 180,E1 -15091.326,E2 -15091.326} C_VEL
LIN {X 0,Y 320.744,Z 415.531,A -85,B 0,C 180,E1 -15092.684,E2 -15092.684} C_VEL
LIN {X 0,Y 319.716,Z 415.658,A -85,B 0,C 180,E1 -15093.736,E2 -15093.736} C_VEL
LIN {X 0,Y 319.634,Z 415.669,A -85,B 0,C 180,E1 -15094.092,E2 -15094.092} C_VEL
LIN {X 0,Y 319.599,Z 415.675,A -85,B 0,C 180,E1 -15098.048,E2 -15098.048} C_VEL
LIN {X 0,Y 319.691,Z 415.66,A -85,B 0,C 180,E1 -15100.962,E2 -15100.962} C_VEL
LIN {X 0,Y 319.734,Z 415.654,A -85,B 0,C 180,E1 -15105.276,E2 -15105.276} C_VEL
LIN {X 0,Y 319.761,Z 415.656,A -85,B 0,C 180,E1 -15109.873,E2 -15109.873} C_VEL
LIN {X 0,Y 319.936,Z 415.631,A -85,B 0,C 180,E1 -15112.426,E2 -15112.426} C_VEL
LIN {X 0,Y 319.749,Z 415.653,A -85,B 0,C 180,E1 -15114.956,E2 -15114.956} C_VEL
LIN {X 0,Y 319.992,Z 415.624,A -85,B 0,C 180,E1 -15117.482,E2 -15117.482} C_VEL
LIN {X 0,Y 320.152,Z 415.607,A -85,B 0,C 180,E1 -15120,E2 -15120} C_VEL
LIN {X 0,Y 319.993,Z 415.622,A -85,B 0,C 180,E1 -15122.518,E2 -15122.518} C_VEL
LIN {X 0,Y 319.955,Z 415.628,A -85,B 0,C 180,E1 -15126.305,E2 -15126.305} C_VEL
LIN {X 0,Y 319.846,Z 415.641,A -85,B 0,C 180,E1 -15128.848,E2 -15128.848} C_VEL
LIN {X 0,Y 319.688,Z 415.661,A -85,B 0,C 180,E1 -15132.7,E2 -15132.7} C_VEL
LIN {X 0,Y 319.702,Z 415.662,A -85,B 0,C 180,E1 -15135.295,E2 -15135.295} C_VEL
LIN {X 0,Y 319.677,Z 415.666,A -85,B 0,C 180,E1 -15139.255,E2 -15139.255} C_VEL
LIN {X 0,Y 319.573,Z 415.68,A -85,B 0,C 180,E1 -15143.319,E2 -15143.319} C_VEL
LIN {X 0,Y 319.62,Z 415.669,A -85,B 0,C 180,E1 -15146.089,E2 -15146.089} C_VEL
LIN {X 0,Y 319.582,Z 415.676,A -85,B 0,C 180,E1 -15148.934,E2 -15148.934} C_VEL
LIN {X 0,Y 319.533,Z 415.678,A -85,B 0,C 180,E1 -15151.862,E2 -15151.862} C_VEL
LIN {X 0,Y 319.582,Z 415.675,A -85,B 0,C 180,E1 -15155.543,E2 -15155.543} C_VEL
LIN {X 0,Y 319.559,Z 415.677,A -85,B 0,C 180,E1 -15158.01,E2 -15158.01} C_VEL
LIN {X 0,Y 319.528,Z 415.685,A -85,B 0,C 180,E1 -15161.597,E2 -15161.597} C_VEL
LIN {X 0,Y 319.557,Z 415.751,A -85,B 0,C 180,E1 -15164.874,E2 -15164.874} C_VEL
LIN {X 0,Y 320.395,Z 420.453,A -85,B 0,C 180,E1 -15168.847,E2 -15168.847} C_VEL
LIN {X 0,Y 321.015,Z 424.717,A -85,B 0,C 180,E1 -15172.193,E2 -15172.193} C_VEL
LIN {X 0,Y 321.174,Z 427.249,A -85,B 0,C 180,E1 -15174.061,E2 -15174.061} C_VEL
LIN {X 0,Y 320.745,Z 431.129,A -85,B 0,C 180,E1 -15176.784,E2 -15176.784} C_VEL
LIN {X 0,Y 320.108,Z 436.402,A -85,B 0,C 180,E1 -15180.397,E2 -15180.397} C_VEL
LIN {X 0,Y 319.4,Z 442.469,A -85,B 0,C 180,E1 -15184.443,E2 -15184.443} C_VEL
LIN {X 0,Y 319.033,Z 446.524,A -85,B 0,C 180,E1 -15187.122,E2 -15187.122} C_VEL
LIN {X 0,Y 322.121,Z 460.3,A -85,B 0,C 180,E1 -15187.923,E2 -15187.923} C_VEL
LIN {X 0,Y 324.311,Z 473.479,A -85,B 0,C 180,E1 -15188.911,E2 -15188.911} C_VEL
LIN {X 0,Y 325.459,Z 484.857,A -85,B 0,C 180,E1 -15189.952,E2 -15189.952} C_VEL
LIN {X 0,Y 325.634,Z 489.727,A -85,B 0,C 180,E1 -15190.456,E2 -15190.456} C_VEL
LIN {X 0,Y 324.231,Z 500.691,A -85,B 0,C 180,E1 -15191.681,E2 -15191.681} C_VEL
LIN {X 0,Y 322.853,Z 510.691,A -85,B 0,C 180,E1 -15193.09,E2 -15193.09} C_VEL
LIN {X 0,Y 321.507,Z 520.411,A -85,B 0,C 180,E1 -15194.792,E2 -15194.792} C_VEL
LIN {X 0,Y 320.437,Z 527.713,A -85,B 0,C 180,E1 -15196.363,E2 -15196.363} C_VEL
LIN {X 0,Y 319.336,Z 534.902,A -85,B 0,C 180,E1 -15198.254,E2 -15198.254} C_VEL
LIN {X 0,Y 318.744,Z 539.76,A -85,B 0,C 180,E1 -15199.84,E2 -15199.84} C_VEL
LIN {X 0,Y 318.23,Z 544.483,A -85,B 0,C 180,E1 -15201.747,E2 -15201.747} C_VEL
LIN {X 0,Y 317.89,Z 548.092,A -85,B 0,C 180,E1 -15203.653,E2 -15203.653} C_VEL
LIN {X 0,Y 317.804,Z 549.955,A -85,B 0,C 180,E1 -15204.925,E2 -15204.925} C_VEL
LIN {X 0,Y 317.808,Z 551.354,A -85,B 0,C 180,E1 -15206.196,E2 -15206.196} C_VEL
LIN {X 0,Y 317.759,Z 552.351,A -85,B 0,C 180,E1 -15207.465,E2 -15207.465} C_VEL
LIN {X 0,Y 317.743,Z 552.959,A -85,B 0,C 180,E1 -15208.732,E2 -15208.732} C_VEL
LIN {X 0,Y 317.782,Z 553.174,A -85,B 0,C 180,E1 -15210,E2 -15210} C_VEL
LIN {X 0,Y 317.743,Z 552.953,A -85,B 0,C 180,E1 -15211.267,E2 -15211.267} C_VEL
LIN {X 0,Y 317.759,Z 552.342,A -85,B 0,C 180,E1 -15212.535,E2 -15212.535} C_VEL
LIN {X 0,Y 317.808,Z 551.343,A -85,B 0,C 180,E1 -15213.804,E2 -15213.804} C_VEL
LIN {X 0,Y 317.831,Z 549.061,A -85,B 0,C 180,E1 -15215.698,E2 -15215.698} C_VEL
LIN {X 0,Y 318.085,Z 545.762,A -85,B 0,C 180,E1 -15217.618,E2 -15217.618} C_VEL
LIN {X 0,Y 318.557,Z 541.412,A -85,B 0,C 180,E1 -15219.524,E2 -15219.524} C_VEL
LIN {X 0,Y 319.21,Z 535.873,A -85,B 0,C 180,E1 -15221.429,E2 -15221.429} C_VEL
LIN {X 0,Y 320.253,Z 528.966,A -85,B 0,C 180,E1 -15223.322,E2 -15223.322} C_VEL
LIN {X 0,Y 321.284,Z 521.913,A -85,B 0,C 180,E1 -15224.894,E2 -15224.894} C_VEL
LIN {X 0,Y 322.594,Z 512.846,A -85,B 0,C 180,E1 -15226.548,E2 -15226.548} C_VEL
LIN {X 0,Y 323.896,Z 502.914,A -85,B 0,C 180,E1 -15228.011,E2 -15228.011} C_VEL
LIN {X 0,Y 325.454,Z 491.099,A -85,B 0,C 180,E1 -15229.391,E2 -15229.391} C_VEL
LIN {X 0,Y 325.443,Z 484.657,A -85,B 0,C 180,E1 -15230.049,E2 -15230.049} C_VEL
LIN {X 0,Y 324.101,Z 472.137,A -85,B 0,C 180,E1 -15231.181,E2 -15231.181} C_VEL
LIN {X 0,Y 321.873,Z 459.107,A -85,B 0,C 180,E1 -15232.138,E2 -15232.138} C_VEL
LIN {X 0,Y 319.017,Z 446.522,A -85,B 0,C 180,E1 -15232.861,E2 -15232.861} C_VEL
LIN {X 0,Y 319.57,Z 440.57,A -85,B 0,C 180,E1 -15236.797,E2 -15236.797} C_VEL
LIN {X 0,Y 320.233,Z 435.298,A -85,B 0,C 180,E1 -15240.316,E2 -15240.316} C_VEL
LIN {X 0,Y 320.86,Z 430.444,A -85,B 0,C 180,E1 -15243.66,E2 -15243.66} C_VEL
LIN {X 0,Y 321.104,Z 426.829,A -85,B 0,C 180,E1 -15246.224,E2 -15246.224} C_VEL
LIN {X 0,Y 321.003,Z 424.441,A -85,B 0,C 180,E1 -15247.984,E2 -15247.984} C_VEL
LIN {X 0,Y 320.403,Z 420.425,A -85,B 0,C 180,E1 -15251.151,E2 -15251.151} C_VEL
LIN {X 0,Y 319.52,Z 415.687,A -85,B 0,C 180,E1 -15255.193,E2 -15255.193} C_VEL
LIN {X 0,Y 319.529,Z 415.685,A -85,B 0,C 180,E1 -15258.712,E2 -15258.712} C_VEL
LIN {X 0,Y 319.563,Z 415.679,A -85,B 0,C 180,E1 -15262.348,E2 -15262.348} C_VEL
LIN {X 0,Y 319.562,Z 415.681,A -85,B 0,C 180,E1 -15265.123,E2 -15265.123} C_VEL
LIN {X 0,Y 319.567,Z 415.68,A -85,B 0,C 180,E1 -15269.059,E2 -15269.059} C_VEL
LIN {X 0,Y 319.607,Z 415.674,A -85,B 0,C 180,E1 -15272.498,E2 -15272.498} C_VEL
LIN {X 0,Y 319.606,Z 415.672,A -85,B 0,C 180,E1 -15275.304,E2 -15275.304} C_VEL
LIN {X 0,Y 319.599,Z 415.673,A -85,B 0,C 180,E1 -15278.048,E2 -15278.048} C_VEL
LIN {X 0,Y 319.69,Z 415.663,A -85,B 0,C 180,E1 -15280.962,E2 -15280.962} C_VEL
LIN {X 0,Y 319.732,Z 415.656,A -85,B 0,C 180,E1 -15285.276,E2 -15285.276} C_VEL
LIN {X 0,Y 319.761,Z 415.653,A -85,B 0,C 180,E1 -15289.873,E2 -15289.873} C_VEL
LIN {X 0,Y 319.935,Z 415.634,A -85,B 0,C 180,E1 -15292.426,E2 -15292.426} C_VEL
LIN {X 0,Y 319.748,Z 415.653,A -85,B 0,C 180,E1 -15294.956,E2 -15294.956} C_VEL
LIN {X 0,Y 319.991,Z 415.623,A -85,B 0,C 180,E1 -15297.482,E2 -15297.482} C_VEL
LIN {X 0,Y 320.17,Z 415.604,A -85,B 0,C 180,E1 -15300,E2 -15300} C_VEL
LIN {X 0,Y 319.991,Z 415.625,A -85,B 0,C 180,E1 -15302.518,E2 -15302.518} C_VEL
LIN {X 0,Y 319.932,Z 415.631,A -85,B 0,C 180,E1 -15306.665,E2 -15306.665} C_VEL
LIN {X 0,Y 319.761,Z 415.656,A -85,B 0,C 180,E1 -15310.127,E2 -15310.127} C_VEL
LIN {X 0,Y 319.732,Z 415.655,A -85,B 0,C 180,E1 -15314.724,E2 -15314.724} C_VEL
LIN {X 0,Y 319.69,Z 415.66,A -85,B 0,C 180,E1 -15319.038,E2 -15319.038} C_VEL
LIN {X 0,Y 319.572,Z 415.676,A -85,B 0,C 180,E1 -15323.319,E2 -15323.319} C_VEL
LIN {X 0,Y 319.635,Z 415.669,A -85,B 0,C 180,E1 -15326.088,E2 -15326.088} C_VEL
LIN {X 0,Y 319.589,Z 415.673,A -85,B 0,C 180,E1 -15328.934,E2 -15328.934} C_VEL
LIN {X 0,Y 319.535,Z 415.682,A -85,B 0,C 180,E1 -15331.862,E2 -15331.862} C_VEL
LIN {X 0,Y 319.582,Z 415.679,A -85,B 0,C 180,E1 -15335.544,E2 -15335.544} C_VEL
LIN {X 0,Y 319.575,Z 415.676,A -85,B 0,C 180,E1 -15338.008,E2 -15338.008} C_VEL
LIN {X 0,Y 319.527,Z 415.685,A -85,B 0,C 180,E1 -15341.597,E2 -15341.597} C_VEL
LIN {X 0,Y 319.517,Z 415.687,A -85,B 0,C 180,E1 -15345.262,E2 -15345.262} C_VEL
LIN {X 0,Y 319.53,Z 415.682,A -85,B 0,C 180,E1 -15348.712,E2 -15348.712} C_VEL
LIN {X 0,Y 319.511,Z 415.687,A -85,B 0,C 180,E1 -15351.983,E2 -15351.983} C_VEL
LIN {X 0,Y 319.547,Z 416.508,A -85,B 0,C 180,E1 -15353.571,E2 -15353.571} C_VEL
LIN {X 0,Y 319.489,Z 419.518,A -85,B 0,C 180,E1 -15356.711,E2 -15356.711} C_VEL
LIN {X 0,Y 319.277,Z 422.426,A -85,B 0,C 180,E1 -15359.584,E2 -15359.584} C_VEL
LIN {X 0,Y 319.045,Z 425.401,A -85,B 0,C 180,E1 -15362.445,E2 -15362.445} C_VEL
LIN {X 0,Y 318.81,Z 428.421,A -85,B 0,C 180,E1 -15365.238,E2 -15365.238} C_VEL
LIN {X 0,Y 318.663,Z 430.577,A -85,B 0,C 180,E1 -15367.173,E2 -15367.173} C_VEL
LIN {X 0,Y 322.935,Z 445.827,A -85,B 0,C 180,E1 -15368.198,E2 -15368.198} C_VEL
LIN {X 0,Y 325.673,Z 458.414,A -85,B 0,C 180,E1 -15369.248,E2 -15369.248} C_VEL
LIN {X 0,Y 326.835,Z 466.559,A -85,B 0,C 180,E1 -15370.04,E2 -15370.04} C_VEL
LIN {X 0,Y 325.685,Z 477.306,A -85,B 0,C 180,E1 -15371.114,E2 -15371.114} C_VEL
LIN {X 0,Y 324.547,Z 487.183,A -85,B 0,C 180,E1 -15372.352,E2 -15372.352} C_VEL
LIN {X 0,Y 323.215,Z 497.15,A -85,B 0,C 180,E1 -15373.905,E2 -15373.905} C_VEL
LIN {X 0,Y 321.885,Z 505.315,A -85,B 0,C 180,E1 -15375.458,E2 -15375.458} C_VEL
LIN {X 0,Y 320.69,Z 513.308,A -85,B 0,C 180,E1 -15377.341,E2 -15377.341} C_VEL
LIN {X 0,Y 319.714,Z 519.723,A -85,B 0,C 180,E1 -15379.231,E2 -15379.231} C_VEL
LIN {X 0,Y 318.895,Z 524.813,A -85,B 0,C 180,E1 -15381.126,E2 -15381.126} C_VEL
LIN {X 0,Y 318.386,Z 529.344,A -85,B 0,C 180,E1 -15383.377,E2 -15383.377} C_VEL
LIN {X 0,Y 318.159,Z 531.674,A -85,B 0,C 180,E1 -15384.931,E2 -15384.931} C_VEL
LIN {X 0,Y 317.991,Z 533.071,A -85,B 0,C 180,E1 -15386.198,E2 -15386.198} C_VEL
LIN {X 0,Y 317.787,Z 534.676,A -85,B 0,C 180,E1 -15388.733,E2 -15388.733} C_VEL
LIN {X 0,Y 317.788,Z 534.907,A -85,B 0,C 180,E1 -15390,E2 -15390} C_VEL
LIN {X 0,Y 317.787,Z 534.716,A -85,B 0,C 180,E1 -15391.267,E2 -15391.267} C_VEL
LIN {X 0,Y 317.987,Z 533.162,A -85,B 0,C 180,E1 -15393.802,E2 -15393.802} C_VEL
LIN {X 0,Y 318.151,Z 531.805,A -85,B 0,C 180,E1 -15395.069,E2 -15395.069} C_VEL
LIN {X 0,Y 318.386,Z 529.52,A -85,B 0,C 180,E1 -15396.623,E2 -15396.623} C_VEL
LIN {X 0,Y 318.892,Z 525.054,A -85,B 0,C 180,E1 -15398.875,E2 -15398.875} C_VEL
LIN {X 0,Y 319.674,Z 520.036,A -85,B 0,C 180,E1 -15400.77,E2 -15400.77} C_VEL
LIN {X 0,Y 320.609,Z 513.719,A -85,B 0,C 180,E1 -15402.663,E2 -15402.663} C_VEL
LIN {X 0,Y 321.827,Z 505.81,A -85,B 0,C 180,E1 -15404.545,E2 -15404.545} C_VEL
LIN {X 0,Y 323.38,Z 495.969,A -85,B 0,C 180,E1 -15406.411,E2 -15406.411} C_VEL
LIN {X 0,Y 324.669,Z 485.641,A -85,B 0,C 180,E1 -15407.967,E2 -15407.967} C_VEL
LIN {X 0,Y 325.929,Z 475.407,A -85,B 0,C 180,E1 -15409.198,E2 -15409.198} C_VEL
LIN {X 0,Y 326.831,Z 465.97,A -85,B 0,C 180,E1 -15410.124,E2 -15410.124} C_VEL
LIN {X 0,Y 324.825,Z 454.2,A -85,B 0,C 180,E1 -15411.238,E2 -15411.238} C_VEL
LIN {X 0,Y 321.918,Z 441.796,A -85,B 0,C 180,E1 -15412.209,E2 -15412.209} C_VEL
LIN {X 0,Y 318.675,Z 430.588,A -85,B 0,C 180,E1 -15412.929,E2 -15412.929} C_VEL
LIN {X 0,Y 318.908,Z 427.024,A -85,B 0,C 180,E1 -15416.152,E2 -15416.152} C_VEL
LIN {X 0,Y 319.15,Z 424.049,A -85,B 0,C 180,E1 -15418.977,E2 -15418.977} C_VEL
LIN {X 0,Y 319.372,Z 421.062,A -85,B 0,C 180,E1 -15421.88,E2 -15421.88} C_VEL
LIN {X 0,Y 319.587,Z 417.447,A -85,B 0,C 180,E1 -15425.544,E2 -15425.544} C_VEL
LIN {X 0,Y 319.514,Z 415.686,A -85,B 0,C 180,E1 -15427.641,E2 -15427.641} C_VEL
LIN {X 0,Y 319.531,Z 415.681,A -85,B 0,C 180,E1 -15431.288,E2 -15431.288} C_VEL
LIN {X 0,Y 319.518,Z 415.686,A -85,B 0,C 180,E1 -15434.738,E2 -15434.738} C_VEL
LIN {X 0,Y 319.528,Z 415.684,A -85,B 0,C 180,E1 -15438.403,E2 -15438.403} C_VEL
LIN {X 0,Y 319.581,Z 415.677,A -85,B 0,C 180,E1 -15442.344,E2 -15442.344} C_VEL
LIN {X 0,Y 319.563,Z 415.677,A -85,B 0,C 180,E1 -15445.124,E2 -15445.124} C_VEL
LIN {X 0,Y 319.573,Z 415.676,A -85,B 0,C 180,E1 -15449.058,E2 -15449.058} C_VEL
LIN {X 0,Y 319.609,Z 415.674,A -85,B 0,C 180,E1 -15452.498,E2 -15452.498} C_VEL
LIN {X 0,Y 319.634,Z 415.669,A -85,B 0,C 180,E1 -15454.092,E2 -15454.092} C_VEL
LIN {X 0,Y 318.962,Z 415.756,A -85,B 0,C 180,E1 -15455.144,E2 -15455.144} C_VEL
LIN {X 0,Y 316.078,Z 416.113,A -85,B 0,C 180,E1 -15456.855,E2 -15456.855} C_VEL
LIN {X 0,Y 313.646,Z 416.418,A -85,B 0,C 180,E1 -15458.243,E2 -15458.243} C_VEL
LIN {X 0,Y 312.625,Z 416.54,A -85,B 0,C 180,E1 -15459.318,E2 -15459.318} C_VEL
LIN {X 0,Y 312.554,Z 416.549,A -85,B 0,C 180,E1 -15459.682,E2 -15459.682} C_VEL
LIN {X 0,Y 312.609,Z 416.542,A -85,B 0,C 180,E1 -15463.006,E2 -15463.006} C_VEL
LIN {X 0,Y 312.696,Z 416.533,A -85,B 0,C 180,E1 -15465.686,E2 -15465.686} C_VEL
LIN {X 0,Y 312.705,Z 416.532,A -85,B 0,C 180,E1 -15469.642,E2 -15469.642} C_VEL
LIN {X 0,Y 312.875,Z 416.512,A -85,B 0,C 180,E1 -15472.254,E2 -15472.254} C_VEL
LIN {X 0,Y 312.72,Z 416.529,A -85,B 0,C 180,E1 -15474.842,E2 -15474.842} C_VEL
LIN {X 0,Y 312.991,Z 416.495,A -85,B 0,C 180,E1 -15478.713,E2 -15478.713} C_VEL
LIN {X 0,Y 312.993,Z 416.496,A -85,B 0,C 180,E1 -15481.287,E2 -15481.287} C_VEL
LIN {X 0,Y 312.72,Z 416.53,A -85,B 0,C 180,E1 -15485.158,E2 -15485.158} C_VEL
LIN {X 0,Y 312.875,Z 416.514,A -85,B 0,C 180,E1 -15487.746,E2 -15487.746} C_VEL
LIN {X 0,Y 312.675,Z 416.539,A -85,B 0,C 180,E1 -15491.671,E2 -15491.671} C_VEL
LIN {X 0,Y 312.703,Z 416.532,A -85,B 0,C 180,E1 -15494.888,E2 -15494.888} C_VEL
LIN {X 0,Y 312.633,Z 416.543,A -85,B 0,C 180,E1 -15499.237,E2 -15499.237} C_VEL
LIN {X 0,Y 312.548,Z 416.551,A -85,B 0,C 180,E1 -15502.789,E2 -15502.789} C_VEL
LIN {X 0,Y 312.599,Z 416.544,A -85,B 0,C 180,E1 -15505.933,E2 -15505.933} C_VEL
LIN {X 0,Y 312.54,Z 416.553,A -85,B 0,C 180,E1 -15509.651,E2 -15509.651} C_VEL
LIN {X 0,Y 312.521,Z 416.554,A -85,B 0,C 180,E1 -15513.689,E2 -15513.689} C_VEL
LIN {X 0,Y 312.528,Z 416.555,A -85,B 0,C 180,E1 -15517.385,E2 -15517.385} C_VEL
LIN {X 0,Y 312.492,Z 416.563,A -85,B 0,C 180,E1 -15520.709,E2 -15520.709} C_VEL
LIN {X 0,Y 312.494,Z 416.596,A -85,B 0,C 180,E1 -15524.427,E2 -15524.427} C_VEL
LIN {X 0,Y 313.173,Z 420.429,A -85,B 0,C 180,E1 -15527.779,E2 -15527.779} C_VEL
LIN {X 0,Y 313.899,Z 425.101,A -85,B 0,C 180,E1 -15531.594,E2 -15531.594} C_VEL
LIN {X 0,Y 314.129,Z 427.77,A -85,B 0,C 180,E1 -15533.652,E2 -15533.652} C_VEL
LIN {X 0,Y 313.865,Z 430.952,A -85,B 0,C 180,E1 -15535.958,E2 -15535.958} C_VEL
LIN {X 0,Y 313.156,Z 436.208,A -85,B 0,C 180,E1 -15539.671,E2 -15539.671} C_VEL
LIN {X 0,Y 312.487,Z 441.454,A -85,B 0,C 180,E1 -15543.268,E2 -15543.268} C_VEL
LIN {X 0,Y 312.009,Z 446.324,A -85,B 0,C 180,E1 -15546.578,E2 -15546.578} C_VEL
LIN {X 0,Y 315.121,Z 459.938,A -85,B 0,C 180,E1 -15547.397,E2 -15547.397} C_VEL
LIN {X 0,Y 317.11,Z 471.448,A -85,B 0,C 180,E1 -15548.271,E2 -15548.271} C_VEL
LIN {X 0,Y 318.48,Z 482.875,A -85,B 0,C 180,E1 -15549.324,E2 -15549.324} C_VEL
LIN {X 0,Y 318.767,Z 491.058,A -85,B 0,C 180,E1 -15550.185,E2 -15550.185} C_VEL
LIN {X 0,Y 317.149,Z 502.845,A -85,B 0,C 180,E1 -15551.592,E2 -15551.592} C_VEL
LIN {X 0,Y 315.672,Z 513.316,A -85,B 0,C 180,E1 -15553.176,E2 -15553.176} C_VEL
LIN {X 0,Y 314.385,Z 521.791,A -85,B 0,C 180,E1 -15554.771,E2 -15554.771} C_VEL
LIN {X 0,Y 313.12,Z 530.066,A -85,B 0,C 180,E1 -15556.699,E2 -15556.699} C_VEL
LIN {X 0,Y 312.094,Z 536.737,A -85,B 0,C 180,E1 -15558.636,E2 -15558.636} C_VEL
LIN {X 0,Y 311.35,Z 542.845,A -85,B 0,C 180,E1 -15560.909,E2 -15560.909} C_VEL
LIN {X 0,Y 310.92,Z 546.816,A -85,B 0,C 180,E1 -15562.858,E2 -15562.858} C_VEL
LIN {X 0,Y 310.708,Z 549.751,A -85,B 0,C 180,E1 -15564.809,E2 -15564.809} C_VEL
LIN {X 0,Y 310.718,Z 551.15,A -85,B 0,C 180,E1 -15566.109,E2 -15566.109} C_VEL
LIN {X 0,Y 310.683,Z 552.147,A -85,B 0,C 180,E1 -15567.407,E2 -15567.407} C_VEL
LIN {X 0,Y 310.658,Z 552.755,A -85,B 0,C 180,E1 -15568.704,E2 -15568.704} C_VEL
LIN {X 0,Y 310.692,Z 552.97,A -85,B 0,C 180,E1 -15570,E2 -15570} C_VEL
LIN {X 0,Y 310.658,Z 552.749,A -85,B 0,C 180,E1 -15571.296,E2 -15571.296} C_VEL
LIN {X 0,Y 310.682,Z 552.138,A -85,B 0,C 180,E1 -15572.593,E2 -15572.593} C_VEL
LIN {X 0,Y 310.718,Z 551.138,A -85,B 0,C 180,E1 -15573.891,E2 -15573.891} C_VEL
LIN {X 0,Y 310.726,Z 549.145,A -85,B 0,C 180,E1 -15575.619,E2 -15575.619} C_VEL
LIN {X 0,Y 311.027,Z 545.556,A -85,B 0,C 180,E1 -15577.792,E2 -15577.792} C_VEL
LIN {X 0,Y 311.51,Z 541.206,A -85,B 0,C 180,E1 -15579.742,E2 -15579.742} C_VEL
LIN {X 0,Y 312.2,Z 535.666,A -85,B 0,C 180,E1 -15581.689,E2 -15581.689} C_VEL
LIN {X 0,Y 313.301,Z 528.759,A -85,B 0,C 180,E1 -15583.623,E2 -15583.623} C_VEL
LIN {X 0,Y 314.386,Z 521.706,A -85,B 0,C 180,E1 -15585.228,E2 -15585.228} C_VEL
LIN {X 0,Y 315.673,Z 513.207,A -85,B 0,C 180,E1 -15586.823,E2 -15586.823} C_VEL
LIN {X 0,Y 317.118,Z 502.705,A -85,B 0,C 180,E1 -15588.41,E2 -15588.41} C_VEL
LIN {X 0,Y 318.742,Z 490.89,A -85,B 0,C 180,E1 -15589.816,E2 -15589.816} C_VEL
LIN {X 0,Y 318.25,Z 480.586,A -85,B 0,C 180,E1 -15590.888,E2 -15590.888} C_VEL
LIN {X 0,Y 316.607,Z 468.189,A -85,B 0,C 180,E1 -15591.971,E2 -15591.971} C_VEL
LIN {X 0,Y 314.134,Z 455.374,A -85,B 0,C 180,E1 -15592.879,E2 -15592.879} C_VEL
LIN {X 0,Y 312.004,Z 446.297,A -85,B 0,C 180,E1 -15593.419,E2 -15593.419} C_VEL
LIN {X 0,Y 312.622,Z 440.375,A -85,B 0,C 180,E1 -15597.442,E2 -15597.442} C_VEL
LIN {X 0,Y 313.344,Z 435.113,A -85,B 0,C 180,E1 -15601.055,E2 -15601.055} C_VEL
LIN {X 0,Y 314.053,Z 429.854,A -85,B 0,C 180,E1 -15604.795,E2 -15604.795} C_VEL
LIN {X 0,Y 314.095,Z 426.644,A -85,B 0,C 180,E1 -15607.167,E2 -15607.167} C_VEL
LIN {X 0,Y 313.55,Z 422.386,A -85,B 0,C 180,E1 -15610.543,E2 -15610.543} C_VEL
LIN {X 0,Y 312.747,Z 418.158,A -85,B 0,C 180,E1 -15614.157,E2 -15614.157} C_VEL
LIN {X 0,Y 312.47,Z 416.565,A -85,B 0,C 180,E1 -15615.681,E2 -15615.681} C_VEL
LIN {X 0,Y 312.491,Z 416.562,A -85,B 0,C 180,E1 -15619.291,E2 -15619.291} C_VEL
LIN {X 0,Y 312.527,Z 416.558,A -85,B 0,C 180,E1 -15622.615,E2 -15622.615} C_VEL
LIN {X 0,Y 312.52,Z 416.556,A -85,B 0,C 180,E1 -15626.311,E2 -15626.311} C_VEL
LIN {X 0,Y 312.539,Z 416.554,A -85,B 0,C 180,E1 -15630.349,E2 -15630.349} C_VEL
LIN {X 0,Y 312.598,Z 416.544,A -85,B 0,C 180,E1 -15634.067,E2 -15634.067} C_VEL
LIN {X 0,Y 312.588,Z 416.546,A -85,B 0,C 180,E1 -15637.529,E2 -15637.529} C_VEL
LIN {X 0,Y 312.64,Z 416.539,A -85,B 0,C 180,E1 -15641.656,E2 -15641.656} C_VEL
LIN {X 0,Y 312.695,Z 416.532,A -85,B 0,C 180,E1 -15645.686,E2 -15645.686} C_VEL
LIN {X 0,Y 312.705,Z 416.531,A -85,B 0,C 180,E1 -15649.642,E2 -15649.642} C_VEL
LIN {X 0,Y 312.874,Z 416.514,A -85,B 0,C 180,E1 -15652.254,E2 -15652.254} C_VEL
LIN {X 0,Y 312.719,Z 416.53,A -85,B 0,C 180,E1 -15654.842,E2 -15654.842} C_VEL
LIN {X 0,Y 312.992,Z 416.496,A -85,B 0,C 180,E1 -15658.713,E2 -15658.713} C_VEL
LIN {X 0,Y 313.122,Z 416.482,A -85,B 0,C 180,E1 -15660,E2 -15660} C_VEL
LIN {X 0,Y 312.937,Z 416.503,A -85,B 0,C 180,E1 -15662.574,E2 -15662.574} C_VEL
LIN {X 0,Y 312.895,Z 416.508,A -85,B 0,C 180,E1 -15666.648,E2 -15666.648} C_VEL
LIN {X 0,Y 312.789,Z 416.52,A -85,B 0,C 180,E1 -15669.049,E2 -15669.049} C_VEL
LIN {X 0,Y 312.639,Z 416.539,A -85,B 0,C 180,E1 -15672.991,E2 -15672.991} C_VEL
LIN {X 0,Y 312.64,Z 416.542,A -85,B 0,C 180,E1 -15675.65,E2 -15675.65} C_VEL
LIN {X 0,Y 312.631,Z 416.539,A -85,B 0,C 180,E1 -15679.236,E2 -15679.236} C_VEL
LIN {X 0,Y 312.547,Z 416.55,A -85,B 0,C 180,E1 -15682.789,E2 -15682.789} C_VEL
LIN {X 0,Y 312.604,Z 416.546,A -85,B 0,C 180,E1 -15685.936,E2 -15685.936} C_VEL
LIN {X 0,Y 312.546,Z 416.555,A -85,B 0,C 180,E1 -15689.65,E2 -15689.65} C_VEL
LIN {X 0,Y 312.521,Z 416.557,A -85,B 0,C 180,E1 -15693.689,E2 -15693.689} C_VEL
LIN {X 0,Y 312.54,Z 416.556,A -85,B 0,C 180,E1 -15697.383,E2 -15697.383} C_VEL
LIN {X 0,Y 312.491,Z 416.558,A -85,B 0,C 180,E1 -15700.709,E2 -15700.709} C_VEL
LIN {X 0,Y 312.474,Z 416.56,A -85,B 0,C 180,E1 -15704.206,E2 -15704.206} C_VEL
LIN {X 0,Y 312.487,Z 416.56,A -85,B 0,C 180,E1 -15707.918,E2 -15707.918} C_VEL
LIN {X 0,Y 312.471,Z 416.564,A -85,B 0,C 180,E1 -15710.967,E2 -15710.967} C_VEL
LIN {X 0,Y 312.45,Z 416.676,A -85,B 0,C 180,E1 -15712.604,E2 -15712.604} C_VEL
LIN {X 0,Y 312.536,Z 418.157,A -85,B 0,C 180,E1 -15714.221,E2 -15714.221} C_VEL
LIN {X 0,Y 312.398,Z 421.121,A -85,B 0,C 180,E1 -15717.321,E2 -15717.321} C_VEL
LIN {X 0,Y 312.081,Z 425.256,A -85,B 0,C 180,E1 -15721.435,E2 -15721.435} C_VEL
LIN {X 0,Y 311.84,Z 428.63,A -85,B 0,C 180,E1 -15724.646,E2 -15724.646} C_VEL
LIN {X 0,Y 311.638,Z 430.769,A -85,B 0,C 180,E1 -15726.616,E2 -15726.616} C_VEL
LIN {X 0,Y 316.181,Z 446.738,A -85,B 0,C 180,E1 -15727.747,E2 -15727.747} C_VEL
LIN {X 0,Y 318.824,Z 459.015,A -85,B 0,C 180,E1 -15728.813,E2 -15728.813} C_VEL
LIN {X 0,Y 320.062,Z 468.504,A -85,B 0,C 180,E1 -15729.767,E2 -15729.767} C_VEL
LIN {X 0,Y 318.64,Z 480.147,A -85,B 0,C 180,E1 -15731.015,E2 -15731.015} C_VEL
LIN {X 0,Y 317.471,Z 490.053,A -85,B 0,C 180,E1 -15732.361,E2 -15732.361} C_VEL
LIN {X 0,Y 316.106,Z 499.132,A -85,B 0,C 180,E1 -15733.864,E2 -15733.864} C_VEL
LIN {X 0,Y 314.815,Z 506.999,A -85,B 0,C 180,E1 -15735.455,E2 -15735.455} C_VEL
LIN {X 0,Y 313.563,Z 514.684,A -85,B 0,C 180,E1 -15737.377,E2 -15737.377} C_VEL
LIN {X 0,Y 312.395,Z 521.738,A -85,B 0,C 180,E1 -15739.632,E2 -15739.632} C_VEL
LIN {X 0,Y 311.697,Z 526.434,A -85,B 0,C 180,E1 -15741.573,E2 -15741.573} C_VEL
LIN {X 0,Y 311.267,Z 530.025,A -85,B 0,C 180,E1 -15743.518,E2 -15743.518} C_VEL
LIN {X 0,Y 311.091,Z 531.879,A -85,B 0,C 180,E1 -15744.815,E2 -15744.815} C_VEL
LIN {X 0,Y 310.928,Z 533.275,A -85,B 0,C 180,E1 -15746.112,E2 -15746.112} C_VEL
LIN {X 0,Y 310.701,Z 534.88,A -85,B 0,C 180,E1 -15748.704,E2 -15748.704} C_VEL
LIN {X 0,Y 310.698,Z 535.111,A -85,B 0,C 180,E1 -15750,E2 -15750} C_VEL
LIN {X 0,Y 310.7,Z 534.919,A -85,B 0,C 180,E1 -15751.296,E2 -15751.296} C_VEL
LIN {X 0,Y 310.923,Z 533.365,A -85,B 0,C 180,E1 -15753.888,E2 -15753.888} C_VEL
LIN {X 0,Y 311.082,Z 532.009,A -85,B 0,C 180,E1 -15755.185,E2 -15755.185} C_VEL
LIN {X 0,Y 311.392,Z 529.144,A -85,B 0,C 180,E1 -15757.13,E2 -15757.13} C_VEL
LIN {X 0,Y 311.868,Z 525.257,A -85,B 0,C 180,E1 -15759.076,E2 -15759.076} C_VEL
LIN {X 0,Y 312.693,Z 520.239,A -85,B 0,C 180,E1 -15761.014,E2 -15761.014} C_VEL
LIN {X 0,Y 313.661,Z 513.922,A -85,B 0,C 180,E1 -15762.948,E2 -15762.948} C_VEL
LIN {X 0,Y 314.966,Z 506.011,A -85,B 0,C 180,E1 -15764.869,E2 -15764.869} C_VEL
LIN {X 0,Y 316.588,Z 496.169,A -85,B 0,C 180,E1 -15766.774,E2 -15766.774} C_VEL
LIN {X 0,Y 317.928,Z 485.841,A -85,B 0,C 180,E1 -15768.361,E2 -15768.361} C_VEL
LIN {X 0,Y 319.231,Z 475.606,A -85,B 0,C 180,E1 -15769.617,E2 -15769.617} C_VEL
LIN {X 0,Y 320.129,Z 467.924,A -85,B 0,C 180,E1 -15770.397,E2 -15770.397} C_VEL
LIN {X 0,Y 318.438,Z 457.082,A -85,B 0,C 180,E1 -15771.482,E2 -15771.482} C_VEL
LIN {X 0,Y 315.71,Z 444.923,A -85,B 0,C 180,E1 -15772.505,E2 -15772.505} C_VEL
LIN {X 0,Y 312.006,Z 432.554,A -85,B 0,C 180,E1 -15773.373,E2 -15773.373} C_VEL
LIN {X 0,Y 311.631,Z 430.791,A -85,B 0,C 180,E1 -15773.48,E2 -15773.48} C_VEL
LIN {X 0,Y 311.916,Z 427.222,A -85,B 0,C 180,E1 -15776.785,E2 -15776.785} C_VEL
LIN {X 0,Y 312.155,Z 424.236,A -85,B 0,C 180,E1 -15779.691,E2 -15779.691} C_VEL
LIN {X 0,Y 312.484,Z 420.26,A -85,B 0,C 180,E1 -15783.679,E2 -15783.679} C_VEL
LIN {X 0,Y 312.567,Z 418.092,A -85,B 0,C 180,E1 -15785.957,E2 -15785.957} C_VEL
LIN {X 0,Y 312.491,Z 416.789,A -85,B 0,C 180,E1 -15787.39,E2 -15787.39} C_VEL
LIN {X 0,Y 312.492,Z 416.56,A -85,B 0,C 180,E1 -15790.709,E2 -15790.709} C_VEL
LIN {X 0,Y 312.476,Z 416.56,A -85,B 0,C 180,E1 -15794.206,E2 -15794.206} C_VEL
LIN {X 0,Y 312.488,Z 416.558,A -85,B 0,C 180,E1 -15797.918,E2 -15797.918} C_VEL
LIN {X 0,Y 312.538,Z 416.551,A -85,B 0,C 180,E1 -15801.91,E2 -15801.91} C_VEL
LIN {X 0,Y 312.509,Z 416.556,A -85,B 0,C 180,E1 -15805.79,E2 -15805.79} C_VEL
LIN {X 0,Y 312.526,Z 416.555,A -85,B 0,C 180,E1 -15808.854,E2 -15808.854} C_VEL
LIN {X 0,Y 312.575,Z 416.547,A -85,B 0,C 180,E1 -15811.825,E2 -15811.825} C_VEL
LIN {X 0,Y 312.588,Z 416.547,A -85,B 0,C 180,E1 -15814.711,E2 -15814.711} C_VEL
LIN {X 0,Y 312.59,Z 416.545,A -85,B 0,C 180,E1 -15817.529,E2 -15817.529} C_VEL
LIN {X 0,Y 312.554,Z 416.549,A -85,B 0,C 180,E1 -15819.682,E2 -15819.682} C_VEL
LIN {X 0,Y 311.947,Z 416.63,A -85,B 0,C 180,E1 -15820.757,E2 -15820.757} C_VEL
LIN {X 0,Y 309.209,Z 416.974,A -85,B 0,C 180,E1 -15822.509,E2 -15822.509} C_VEL
LIN {X 0,Y 306.832,Z 417.269,A -85,B 0,C 180,E1 -15823.93,E2 -15823.93} C_VEL
LIN {X 0,Y 305.76,Z 417.397,A -85,B 0,C 180,E1 -15825.028,E2 -15825.028} C_VEL
LIN {X 0,Y 305.646,Z 417.409,A -85,B 0,C 180,E1 -15825.4,E2 -15825.4} C_VEL
LIN {X 0,Y 305.641,Z 417.411,A -85,B 0,C 180,E1 -15829.4,E2 -15829.4} C_VEL
LIN {X 0,Y 305.816,Z 417.393,A -85,B 0,C 180,E1 -15832.074,E2 -15832.074} C_VEL
LIN {X 0,Y 305.691,Z 417.404,A -85,B 0,C 180,E1 -15834.723,E2 -15834.723} C_VEL
LIN {X 0,Y 305.958,Z 417.371,A -85,B 0,C 180,E1 -15838.684,E2 -15838.684} C_VEL
LIN {X 0,Y 305.96,Z 417.372,A -85,B 0,C 180,E1 -15841.316,E2 -15841.316} C_VEL
LIN {X 0,Y 305.855,Z 417.384,A -85,B 0,C 180,E1 -15846.597,E2 -15846.597} C_VEL
LIN {X 0,Y 305.739,Z 417.4,A -85,B 0,C 180,E1 -15849.26,E2 -15849.26} C_VEL
LIN {X 0,Y 305.594,Z 417.419,A -85,B 0,C 180,E1 -15853.296,E2 -15853.296} C_VEL
LIN {X 0,Y 305.596,Z 417.417,A -85,B 0,C 180,E1 -15856.02,E2 -15856.02} C_VEL
LIN {X 0,Y 305.579,Z 417.423,A -85,B 0,C 180,E1 -15859.445,E2 -15859.445} C_VEL
LIN {X 0,Y 305.493,Z 417.431,A -85,B 0,C 180,E1 -15863.041,E2 -15863.041} C_VEL
LIN {X 0,Y 305.528,Z 417.425,A -85,B 0,C 180,E1 -15866.219,E2 -15866.219} C_VEL
LIN {X 0,Y 305.49,Z 417.431,A -85,B 0,C 180,E1 -15869.047,E2 -15869.047} C_VEL
LIN {X 0,Y 305.444,Z 417.432,A -85,B 0,C 180,E1 -15871.952,E2 -15871.952} C_VEL
LIN {X 0,Y 305.465,Z 417.437,A -85,B 0,C 180,E1 -15875.113,E2 -15875.113} C_VEL
LIN {X 0,Y 305.451,Z 417.436,A -85,B 0,C 180,E1 -15878.529,E2 -15878.529} C_VEL
LIN {X 0,Y 305.463,Z 417.439,A -85,B 0,C 180,E1 -15882.587,E2 -15882.587} C_VEL
LIN {X 0,Y 305.502,Z 417.572,A -85,B 0,C 180,E1 -15884.086,E2 -15884.086} C_VEL
LIN {X 0,Y 306.259,Z 422.281,A -85,B 0,C 180,E1 -15888.28,E2 -15888.28} C_VEL
LIN {X 0,Y 306.921,Z 426.507,A -85,B 0,C 180,E1 -15891.811,E2 -15891.811} C_VEL
LIN {X 0,Y 307.081,Z 429.706,A -85,B 0,C 180,E1 -15894.295,E2 -15894.295} C_VEL
LIN {X 0,Y 306.706,Z 432.875,A -85,B 0,C 180,E1 -15896.636,E2 -15896.636} C_VEL
LIN {X 0,Y 305.903,Z 438.697,A -85,B 0,C 180,E1 -15900.813,E2 -15900.813} C_VEL
LIN {X 0,Y 305.189,Z 444.348,A -85,B 0,C 180,E1 -15904.784,E2 -15904.784} C_VEL
LIN {X 0,Y 305.013,Z 446.096,A -85,B 0,C 180,E1 -15906,E2 -15906} C_VEL
LIN {X 0,Y 308.283,Z 460.143,A -85,B 0,C 180,E1 -15906.891,E2 -15906.891} C_VEL
LIN {X 0,Y 310.364,Z 472.214,A -85,B 0,C 180,E1 -15907.849,E2 -15907.849} C_VEL
LIN {X 0,Y 311.572,Z 482.667,A -85,B 0,C 180,E1 -15908.844,E2 -15908.844} C_VEL
LIN {X 0,Y 312.054,Z 490.857,A -85,B 0,C 180,E1 -15909.74,E2 -15909.74} C_VEL
LIN {X 0,Y 310.566,Z 501.466,A -85,B 0,C 180,E1 -15911.016,E2 -15911.016} C_VEL
LIN {X 0,Y 309.097,Z 511.165,A -85,B 0,C 180,E1 -15912.466,E2 -15912.466} C_VEL
LIN {X 0,Y 307.798,Z 520.007,A -85,B 0,C 180,E1 -15914.098,E2 -15914.098} C_VEL
LIN {X 0,Y 306.631,Z 527.308,A -85,B 0,C 180,E1 -15915.736,E2 -15915.736} C_VEL
LIN {X 0,Y 305.391,Z 534.495,A -85,B 0,C 180,E1 -15917.709,E2 -15917.709} C_VEL
LIN {X 0,Y 304.706,Z 539.353,A -85,B 0,C 180,E1 -15919.367,E2 -15919.367} C_VEL
LIN {X 0,Y 304.146,Z 544.076,A -85,B 0,C 180,E1 -15921.361,E2 -15921.361} C_VEL
LIN {X 0,Y 303.74,Z 547.684,A -85,B 0,C 180,E1 -15923.356,E2 -15923.356} C_VEL
LIN {X 0,Y 303.638,Z 549.548,A -85,B 0,C 180,E1 -15924.688,E2 -15924.688} C_VEL
LIN {X 0,Y 303.631,Z 550.946,A -85,B 0,C 180,E1 -15926.018,E2 -15926.018} C_VEL
LIN {X 0,Y 303.607,Z 551.944,A -85,B 0,C 180,E1 -15927.346,E2 -15927.346} C_VEL
LIN {X 0,Y 303.574,Z 552.552,A -85,B 0,C 180,E1 -15928.673,E2 -15928.673} C_VEL
LIN {X 0,Y 303.605,Z 552.767,A -85,B 0,C 180,E1 -15930,E2 -15930} C_VEL
LIN {X 0,Y 303.574,Z 552.545,A -85,B 0,C 180,E1 -15931.326,E2 -15931.326} C_VEL
LIN {X 0,Y 303.607,Z 551.934,A -85,B 0,C 180,E1 -15932.653,E2 -15932.653} C_VEL
LIN {X 0,Y 303.631,Z 550.933,A -85,B 0,C 180,E1 -15933.982,E2 -15933.982} C_VEL
LIN {X 0,Y 303.622,Z 549.229,A -85,B 0,C 180,E1 -15935.538,E2 -15935.538} C_VEL
LIN {X 0,Y 303.991,Z 545.351,A -85,B 0,C 180,E1 -15937.973,E2 -15937.973} C_VEL
LIN {X 0,Y 304.471,Z 540.999,A -85,B 0,C 180,E1 -15939.969,E2 -15939.969} C_VEL
LIN {X 0,Y 305.207,Z 535.459,A -85,B 0,C 180,E1 -15941.961,E2 -15941.961} C_VEL
LIN {X 0,Y 306.381,Z 528.552,A -85,B 0,C 180,E1 -15943.937,E2 -15943.937} C_VEL
LIN {X 0,Y 307.807,Z 519.909,A -85,B 0,C 180,E1 -15945.902,E2 -15945.902} C_VEL
LIN {X 0,Y 309.106,Z 511.045,A -85,B 0,C 180,E1 -15947.533,E2 -15947.533} C_VEL
LIN {X 0,Y 310.547,Z 501.321,A -85,B 0,C 180,E1 -15948.985,E2 -15948.985} C_VEL
LIN {X 0,Y 312.016,Z 490.68,A -85,B 0,C 180,E1 -15950.262,E2 -15950.262} C_VEL
LIN {X 0,Y 311.233,Z 479.074,A -85,B 0,C 180,E1 -15951.496,E2 -15951.496} C_VEL
LIN {X 0,Y 309.585,Z 467.133,A -85,B 0,C 180,E1 -15952.553,E2 -15952.553} C_VEL
LIN {X 0,Y 306.954,Z 454.092,A -85,B 0,C 180,E1 -15953.497,E2 -15953.497} C_VEL
LIN {X 0,Y 305.005,Z 446.055,A -85,B 0,C 180,E1 -15954.006,E2 -15954.006} C_VEL
LIN {X 0,Y 305.698,Z 440.179,A -85,B 0,C 180,E1 -15958.118,E2 -15958.118} C_VEL
LIN {X 0,Y 306.454,Z 434.779,A -85,B 0,C 180,E1 -15961.947,E2 -15961.947} C_VEL
LIN {X 0,Y 307.052,Z 430.737,A -85,B 0,C 180,E1 -15964.905,E2 -15964.905} C_VEL
LIN {X 0,Y 307.068,Z 428.286,A -85,B 0,C 180,E1 -15966.768,E2 -15966.768} C_VEL
LIN {X 0,Y 306.663,Z 424.354,A -85,B 0,C 180,E1 -15969.918,E2 -15969.918} C_VEL
LIN {X 0,Y 305.886,Z 420.096,A -85,B 0,C 180,E1 -15973.573,E2 -15973.573} C_VEL
LIN {X 0,Y 305.42,Z 417.444,A -85,B 0,C 180,E1 -15976.126,E2 -15976.126} C_VEL
LIN {X 0,Y 305.459,Z 417.436,A -85,B 0,C 180,E1 -15979.892,E2 -15979.892} C_VEL
LIN {X 0,Y 305.482,Z 417.434,A -85,B 0,C 180,E1 -15983.631,E2 -15983.631} C_VEL
LIN {X 0,Y 305.466,Z 417.436,A -85,B 0,C 180,E1 -15986.483,E2 -15986.483} C_VEL
LIN {X 0,Y 305.459,Z 417.434,A -85,B 0,C 180,E1 -15989.59,E2 -15989.59} C_VEL
LIN {X 0,Y 305.516,Z 417.43,A -85,B 0,C 180,E1 -15992.608,E2 -15992.608} C_VEL
LIN {X 0,Y 305.509,Z 417.427,A -85,B 0,C 180,E1 -15995.539,E2 -15995.539} C_VEL
LIN {X 0,Y 305.521,Z 417.426,A -85,B 0,C 180,E1 -15999.815,E2 -15999.815} C_VEL
LIN {X 0,Y 305.576,Z 417.424,A -85,B 0,C 180,E1 -16002.603,E2 -16002.603} C_VEL
LIN {X 0,Y 305.65,Z 417.41,A -85,B 0,C 180,E1 -16005.349,E2 -16005.349} C_VEL
LIN {X 0,Y 305.642,Z 417.41,A -85,B 0,C 180,E1 -16009.4,E2 -16009.4} C_VEL
LIN {X 0,Y 305.814,Z 417.392,A -85,B 0,C 180,E1 -16012.074,E2 -16012.074} C_VEL
LIN {X 0,Y 305.69,Z 417.406,A -85,B 0,C 180,E1 -16014.724,E2 -16014.724} C_VEL
LIN {X 0,Y 305.959,Z 417.373,A -85,B 0,C 180,E1 -16018.684,E2 -16018.684} C_VEL
LIN {X 0,Y 305.959,Z 417.371,A -85,B 0,C 180,E1 -16021.316,E2 -16021.316} C_VEL
LIN {X 0,Y 305.851,Z 417.385,A -85,B 0,C 180,E1 -16026.627,E2 -16026.627} C_VEL
LIN {X 0,Y 305.737,Z 417.399,A -85,B 0,C 180,E1 -16029.26,E2 -16029.26} C_VEL
LIN {X 0,Y 305.592,Z 417.417,A -85,B 0,C 180,E1 -16033.296,E2 -16033.296} C_VEL
LIN {X 0,Y 305.595,Z 417.421,A -85,B 0,C 180,E1 -16036.02,E2 -16036.02} C_VEL
LIN {X 0,Y 305.578,Z 417.419,A -85,B 0,C 180,E1 -16039.445,E2 -16039.445} C_VEL
LIN {X 0,Y 305.492,Z 417.429,A -85,B 0,C 180,E1 -16043.042,E2 -16043.042} C_VEL
LIN {X 0,Y 305.533,Z 417.425,A -85,B 0,C 180,E1 -16046.221,E2 -16046.221} C_VEL
LIN {X 0,Y 305.496,Z 417.429,A -85,B 0,C 180,E1 -16049.05,E2 -16049.05} C_VEL
LIN {X 0,Y 305.446,Z 417.437,A -85,B 0,C 180,E1 -16051.952,E2 -16051.952} C_VEL
LIN {X 0,Y 305.464,Z 417.434,A -85,B 0,C 180,E1 -16055.113,E2 -16055.113} C_VEL
LIN {X 0,Y 305.469,Z 417.432,A -85,B 0,C 180,E1 -16058.533,E2 -16058.533} C_VEL
LIN {X 0,Y 305.46,Z 417.434,A -85,B 0,C 180,E1 -16062.587,E2 -16062.587} C_VEL
LIN {X 0,Y 305.444,Z 417.437,A -85,B 0,C 180,E1 -16066.348,E2 -16066.348} C_VEL
LIN {X 0,Y 305.458,Z 417.436,A -85,B 0,C 180,E1 -16069.892,E2 -16069.892} C_VEL
LIN {X 0,Y 305.426,Z 417.443,A -85,B 0,C 180,E1 -16071.59,E2 -16071.59} C_VEL
LIN {X 0,Y 305.489,Z 418.667,A -85,B 0,C 180,E1 -16073.63,E2 -16073.63} C_VEL
LIN {X 0,Y 305.427,Z 421.302,A -85,B 0,C 180,E1 -16076.479,E2 -16076.479} C_VEL
LIN {X 0,Y 305.181,Z 424.303,A -85,B 0,C 180,E1 -16079.56,E2 -16079.56} C_VEL
LIN {X 0,Y 304.915,Z 427.299,A -85,B 0,C 180,E1 -16082.55,E2 -16082.55} C_VEL
LIN {X 0,Y 304.628,Z 431.013,A -85,B 0,C 180,E1 -16086.074,E2 -16086.074} C_VEL
LIN {X 0,Y 308.486,Z 444.186,A -85,B 0,C 180,E1 -16086.997,E2 -16086.997} C_VEL
LIN {X 0,Y 311.354,Z 456.427,A -85,B 0,C 180,E1 -16088.051,E2 -16088.051} C_VEL
LIN {X 0,Y 313.143,Z 466.991,A -85,B 0,C 180,E1 -16089.128,E2 -16089.128} C_VEL
LIN {X 0,Y 313.077,Z 471.874,A -85,B 0,C 180,E1 -16089.638,E2 -16089.638} C_VEL
LIN {X 0,Y 311.609,Z 482.922,A -85,B 0,C 180,E1 -16090.911,E2 -16090.911} C_VEL
LIN {X 0,Y 310.339,Z 493.081,A -85,B 0,C 180,E1 -16092.411,E2 -16092.411} C_VEL
LIN {X 0,Y 308.7,Z 502.652,A -85,B 0,C 180,E1 -16094.145,E2 -16094.145} C_VEL
LIN {X 0,Y 307.25,Z 511.269,A -85,B 0,C 180,E1 -16096.103,E2 -16096.103} C_VEL
LIN {X 0,Y 306.074,Z 518.138,A -85,B 0,C 180,E1 -16098.074,E2 -16098.074} C_VEL
LIN {X 0,Y 305.126,Z 523.636,A -85,B 0,C 180,E1 -16100.052,E2 -16100.052} C_VEL
LIN {X 0,Y 304.493,Z 527.949,A -85,B 0,C 180,E1 -16102.04,E2 -16102.04} C_VEL
LIN {X 0,Y 304.195,Z 530.351,A -85,B 0,C 180,E1 -16103.443,E2 -16103.443} C_VEL
LIN {X 0,Y 304.026,Z 532.084,A -85,B 0,C 180,E1 -16104.695,E2 -16104.695} C_VEL
LIN {X 0,Y 303.867,Z 533.479,A -85,B 0,C 180,E1 -16106.021,E2 -16106.021} C_VEL
LIN {X 0,Y 303.617,Z 535.084,A -85,B 0,C 180,E1 -16108.674,E2 -16108.674} C_VEL
LIN {X 0,Y 303.611,Z 535.314,A -85,B 0,C 180,E1 -16110,E2 -16110} C_VEL
LIN {X 0,Y 303.617,Z 535.123,A -85,B 0,C 180,E1 -16111.327,E2 -16111.327} C_VEL
LIN {X 0,Y 303.862,Z 533.568,A -85,B 0,C 180,E1 -16113.979,E2 -16113.979} C_VEL
LIN {X 0,Y 304.017,Z 532.212,A -85,B 0,C 180,E1 -16115.306,E2 -16115.306} C_VEL
LIN {X 0,Y 304.346,Z 529.346,A -85,B 0,C 180,E1 -16117.297,E2 -16117.297} C_VEL
LIN {X 0,Y 304.845,Z 525.46,A -85,B 0,C 180,E1 -16119.287,E2 -16119.287} C_VEL
LIN {X 0,Y 305.705,Z 520.442,A -85,B 0,C 180,E1 -16121.269,E2 -16121.269} C_VEL
LIN {X 0,Y 306.727,Z 514.124,A -85,B 0,C 180,E1 -16123.246,E2 -16123.246} C_VEL
LIN {X 0,Y 308.12,Z 506.213,A -85,B 0,C 180,E1 -16125.207,E2 -16125.207} C_VEL
LIN {X 0,Y 309.808,Z 496.37,A -85,B 0,C 180,E1 -16127.152,E2 -16127.152} C_VEL
LIN {X 0,Y 311.198,Z 486.041,A -85,B 0,C 180,E1 -16128.773,E2 -16128.773} C_VEL
LIN {X 0,Y 312.576,Z 475.804,A -85,B 0,C 180,E1 -16130.053,E2 -16130.053} C_VEL
LIN {X 0,Y 313.344,Z 469.744,A -85,B 0,C 180,E1 -16130.687,E2 -16130.687} C_VEL
LIN {X 0,Y 311.8,Z 458.617,A -85,B 0,C 180,E1 -16131.856,E2 -16131.856} C_VEL
LIN {X 0,Y 309.09,Z 446.349,A -85,B 0,C 180,E1 -16132.943,E2 -16132.943} C_VEL
LIN {X 0,Y 305.287,Z 433.55,A -85,B 0,C 180,E1 -16133.887,E2 -16133.887} C_VEL
LIN {X 0,Y 304.617,Z 430.964,A -85,B 0,C 180,E1 -16134.09,E2 -16134.09} C_VEL
LIN {X 0,Y 304.916,Z 427.421,A -85,B 0,C 180,E1 -16137.451,E2 -16137.451} C_VEL
LIN {X 0,Y 305.173,Z 424.423,A -85,B 0,C 180,E1 -16140.441,E2 -16140.441} C_VEL
LIN {X 0,Y 305.473,Z 420.893,A -85,B 0,C 180,E1 -16144.08,E2 -16144.08} C_VEL
LIN {X 0,Y 305.486,Z 418.452,A -85,B 0,C 180,E1 -16146.738,E2 -16146.738} C_VEL
LIN {X 0,Y 305.417,Z 417.442,A -85,B 0,C 180,E1 -16148.521,E2 -16148.521} C_VEL
LIN {X 0,Y 305.444,Z 417.434,A -85,B 0,C 180,E1 -16151.857,E2 -16151.857} C_VEL
LIN {X 0,Y 305.421,Z 417.438,A -85,B 0,C 180,E1 -16155.507,E2 -16155.507} C_VEL
LIN {X 0,Y 305.457,Z 417.433,A -85,B 0,C 180,E1 -16159.4,E2 -16159.4} C_VEL
LIN {X 0,Y 305.499,Z 417.429,A -85,B 0,C 180,E1 -16163.264,E2 -16163.264} C_VEL
LIN {X 0,Y 305.467,Z 417.436,A -85,B 0,C 180,E1 -16166.483,E2 -16166.483} C_VEL
LIN {X 0,Y 305.465,Z 417.432,A -85,B 0,C 180,E1 -16169.591,E2 -16169.591} C_VEL
LIN {X 0,Y 305.522,Z 417.428,A -85,B 0,C 180,E1 -16172.609,E2 -16172.609} C_VEL
LIN {X 0,Y 305.51,Z 417.426,A -85,B 0,C 180,E1 -16175.539,E2 -16175.539} C_VEL
LIN {X 0,Y 305.521,Z 417.427,A -85,B 0,C 180,E1 -16179.815,E2 -16179.815} C_VEL
LIN {X 0,Y 305.577,Z 417.42,A -85,B 0,C 180,E1 -16182.603,E2 -16182.603} C_VEL
LIN {X 0,Y 305.646,Z 417.409,A -85,B 0,C 180,E1 -16185.4,E2 -16185.4} C_VEL
LIN {X 0,Y 304.931,Z 417.501,A -85,B 0,C 180,E1 -16186.499,E2 -16186.499} C_VEL
LIN {X 0,Y 302.155,Z 417.848,A -85,B 0,C 180,E1 -16188.293,E2 -16188.293} C_VEL
LIN {X 0,Y 299.839,Z 418.136,A -85,B 0,C 180,E1 -16189.747,E2 -16189.747} C_VEL
LIN {X 0,Y 298.844,Z 418.257,A -85,B 0,C 180,E1 -16190.871,E2 -16190.871} C_VEL
LIN {X 0,Y 298.759,Z 418.267,A -85,B 0,C 180,E1 -16191.251,E2 -16191.251} C_VEL
LIN {X 0,Y 298.801,Z 418.263,A -85,B 0,C 180,E1 -16193.246,E2 -16193.246} C_VEL
LIN {X 0,Y 298.925,Z 418.247,A -85,B 0,C 180,E1 -16198.653,E2 -16198.653} C_VEL
LIN {X 0,Y 298.926,Z 418.249,A -85,B 0,C 180,E1 -16201.347,E2 -16201.347} C_VEL
LIN {X 0,Y 298.801,Z 418.263,A -85,B 0,C 180,E1 -16206.754,E2 -16206.754} C_VEL
LIN {X 0,Y 298.684,Z 418.281,A -85,B 0,C 180,E1 -16209.48,E2 -16209.48} C_VEL
LIN {X 0,Y 298.557,Z 418.297,A -85,B 0,C 180,E1 -16213.615,E2 -16213.615} C_VEL
LIN {X 0,Y 298.551,Z 418.294,A -85,B 0,C 180,E1 -16216.409,E2 -16216.409} C_VEL
LIN {X 0,Y 298.514,Z 418.301,A -85,B 0,C 180,E1 -16219.655,E2 -16219.655} C_VEL
LIN {X 0,Y 298.46,Z 418.308,A -85,B 0,C 180,E1 -16223.597,E2 -16223.597} C_VEL
LIN {X 0,Y 298.487,Z 418.302,A -85,B 0,C 180,E1 -16226.575,E2 -16226.575} C_VEL
LIN {X 0,Y 298.419,Z 418.313,A -85,B 0,C 180,E1 -16229.641,E2 -16229.641} C_VEL
LIN {X 0,Y 298.397,Z 418.31,A -85,B 0,C 180,E1 -16232.8,E2 -16232.8} C_VEL
LIN {X 0,Y 298.448,Z 418.309,A -85,B 0,C 180,E1 -16236.808,E2 -16236.808} C_VEL
LIN {X 0,Y 298.39,Z 418.32,A -85,B 0,C 180,E1 -16241.088,E2 -16241.088} C_VEL
LIN {X 0,Y 298.427,Z 418.333,A -85,B 0,C 180,E1 -16243.538,E2 -16243.538} C_VEL
LIN {X 0,Y 299.068,Z 422.13,A -85,B 0,C 180,E1 -16247.039,E2 -16247.039} C_VEL
LIN {X 0,Y 299.761,Z 426.356,A -85,B 0,C 180,E1 -16250.726,E2 -16250.726} C_VEL
LIN {X 0,Y 300.07,Z 430.591,A -85,B 0,C 180,E1 -16254.159,E2 -16254.159} C_VEL
LIN {X 0,Y 299.678,Z 433.74,A -85,B 0,C 180,E1 -16256.556,E2 -16256.556} C_VEL
LIN {X 0,Y 298.893,Z 439.034,A -85,B 0,C 180,E1 -16260.458,E2 -16260.458} C_VEL
LIN {X 0,Y 298.313,Z 443.303,A -85,B 0,C 180,E1 -16263.541,E2 -16263.541} C_VEL
LIN {X 0,Y 298.017,Z 445.961,A -85,B 0,C 180,E1 -16265.412,E2 -16265.412} C_VEL
LIN {X 0,Y 301.244,Z 459.366,A -85,B 0,C 180,E1 -16266.285,E2 -16266.285} C_VEL
LIN {X 0,Y 303.499,Z 472.111,A -85,B 0,C 180,E1 -16267.329,E2 -16267.329} C_VEL
LIN {X 0,Y 304.742,Z 482.462,A -85,B 0,C 180,E1 -16268.346,E2 -16268.346} C_VEL
LIN {X 0,Y 305.207,Z 492.086,A -85,B 0,C 180,E1 -16269.441,E2 -16269.441} C_VEL
LIN {X 0,Y 303.487,Z 503.619,A -85,B 0,C 180,E1 -16270.907,E2 -16270.907} C_VEL
LIN {X 0,Y 302.023,Z 512.91,A -85,B 0,C 180,E1 -16272.392,E2 -16272.392} C_VEL
LIN {X 0,Y 300.666,Z 521.386,A -85,B 0,C 180,E1 -16274.058,E2 -16274.058} C_VEL
LIN {X 0,Y 299.246,Z 529.66,A -85,B 0,C 180,E1 -16276.07,E2 -16276.07} C_VEL
LIN {X 0,Y 298.099,Z 536.329,A -85,B 0,C 180,E1 -16278.095,E2 -16278.095} C_VEL
LIN {X 0,Y 297.264,Z 542.437,A -85,B 0,C 180,E1 -16280.474,E2 -16280.474} C_VEL
LIN {X 0,Y 296.795,Z 546.408,A -85,B 0,C 180,E1 -16282.517,E2 -16282.517} C_VEL
LIN {X 0,Y 296.552,Z 549.344,A -85,B 0,C 180,E1 -16284.56,E2 -16284.56} C_VEL
LIN {X 0,Y 296.528,Z 550.742,A -85,B 0,C 180,E1 -16285.923,E2 -16285.923} C_VEL
LIN {X 0,Y 296.534,Z 551.741,A -85,B 0,C 180,E1 -16287.283,E2 -16287.283} C_VEL
LIN {X 0,Y 296.494,Z 552.348,A -85,B 0,C 180,E1 -16288.642,E2 -16288.642} C_VEL
LIN {X 0,Y 296.52,Z 552.563,A -85,B 0,C 180,E1 -16290,E2 -16290} C_VEL
LIN {X 0,Y 296.494,Z 552.342,A -85,B 0,C 180,E1 -16291.358,E2 -16291.358} C_VEL
LIN {X 0,Y 296.534,Z 551.731,A -85,B 0,C 180,E1 -16292.717,E2 -16292.717} C_VEL
LIN {X 0,Y 296.528,Z 550.728,A -85,B 0,C 180,E1 -16294.077,E2 -16294.077} C_VEL
LIN {X 0,Y 296.546,Z 549.237,A -85,B 0,C 180,E1 -16295.508,E2 -16295.508} C_VEL
LIN {X 0,Y 296.795,Z 546.376,A -85,B 0,C 180,E1 -16297.483,E2 -16297.483} C_VEL
LIN {X 0,Y 297.264,Z 542.392,A -85,B 0,C 180,E1 -16299.526,E2 -16299.526} C_VEL
LIN {X 0,Y 298.099,Z 536.266,A -85,B 0,C 180,E1 -16301.905,E2 -16301.905} C_VEL
LIN {X 0,Y 299.246,Z 529.583,A -85,B 0,C 180,E1 -16303.929,E2 -16303.929} C_VEL
LIN {X 0,Y 300.671,Z 521.292,A -85,B 0,C 180,E1 -16305.941,E2 -16305.941} C_VEL
LIN {X 0,Y 302.027,Z 512.791,A -85,B 0,C 180,E1 -16307.608,E2 -16307.608} C_VEL
LIN {X 0,Y 303.442,Z 503.465,A -85,B 0,C 180,E1 -16309.096,E2 -16309.096} C_VEL
LIN {X 0,Y 305.167,Z 491.902,A -85,B 0,C 180,E1 -16310.561,E2 -16310.561} C_VEL
LIN {X 0,Y 304.707,Z 482.227,A -85,B 0,C 180,E1 -16311.656,E2 -16311.656} C_VEL
LIN {X 0,Y 303.167,Z 469.758,A -85,B 0,C 180,E1 -16312.858,E2 -16312.858} C_VEL
LIN {X 0,Y 300.627,Z 456.63,A -85,B 0,C 180,E1 -16313.885,E2 -16313.885} C_VEL
LIN {X 0,Y 298.009,Z 445.902,A -85,B 0,C 180,E1 -16314.572,E2 -16314.572} C_VEL
LIN {X 0,Y 298.809,Z 440.005,A -85,B 0,C 180,E1 -16318.808,E2 -16318.808} C_VEL
LIN {X 0,Y 299.515,Z 434.736,A -85,B 0,C 180,E1 -16322.662,E2 -16322.662} C_VEL
LIN {X 0,Y 300.004,Z 431.73,A -85,B 0,C 180,E1 -16324.923,E2 -16324.923} C_VEL
LIN {X 0,Y 299.897,Z 427.368,A -85,B 0,C 180,E1 -16328.391,E2 -16328.391} C_VEL
LIN {X 0,Y 299.372,Z 423.931,A -85,B 0,C 180,E1 -16331.303,E2 -16331.303} C_VEL
LIN {X 0,Y 298.637,Z 419.733,A -85,B 0,C 180,E1 -16335.089,E2 -16335.089} C_VEL
LIN {X 0,Y 298.393,Z 418.317,A -85,B 0,C 180,E1 -16336.456,E2 -16336.456} C_VEL
LIN {X 0,Y 298.404,Z 418.317,A -85,B 0,C 180,E1 -16340.513,E2 -16340.513} C_VEL
LIN {X 0,Y 298.42,Z 418.313,A -85,B 0,C 180,E1 -16343.93,E2 -16343.93} C_VEL
LIN {X 0,Y 298.394,Z 418.315,A -85,B 0,C 180,E1 -16347.984,E2 -16347.984} C_VEL
LIN {X 0,Y 298.458,Z 418.306,A -85,B 0,C 180,E1 -16351.904,E2 -16351.904} C_VEL
LIN {X 0,Y 298.484,Z 418.306,A -85,B 0,C 180,E1 -16354.924,E2 -16354.924} C_VEL
LIN {X 0,Y 298.452,Z 418.307,A -85,B 0,C 180,E1 -16359.315,E2 -16359.315} C_VEL
LIN {X 0,Y 298.539,Z 418.298,A -85,B 0,C 180,E1 -16362.179,E2 -16362.179} C_VEL
LIN {X 0,Y 298.595,Z 418.29,A -85,B 0,C 180,E1 -16364.995,E2 -16364.995} C_VEL
LIN {X 0,Y 298.597,Z 418.289,A -85,B 0,C 180,E1 -16369.147,E2 -16369.147} C_VEL
LIN {X 0,Y 298.76,Z 418.269,A -85,B 0,C 180,E1 -16371.886,E2 -16371.886} C_VEL
LIN {X 0,Y 298.661,Z 418.282,A -85,B 0,C 180,E1 -16374.599,E2 -16374.599} C_VEL
LIN {X 0,Y 298.925,Z 418.249,A -85,B 0,C 180,E1 -16378.653,E2 -16378.653} C_VEL
LIN {X 0,Y 298.925,Z 418.247,A -85,B 0,C 180,E1 -16381.347,E2 -16381.347} C_VEL
LIN {X 0,Y 298.799,Z 418.263,A -85,B 0,C 180,E1 -16386.754,E2 -16386.754} C_VEL
LIN {X 0,Y 298.682,Z 418.278,A -85,B 0,C 180,E1 -16389.48,E2 -16389.48} C_VEL
LIN {X 0,Y 298.555,Z 418.295,A -85,B 0,C 180,E1 -16393.615,E2 -16393.615} C_VEL
LIN {X 0,Y 298.55,Z 418.295,A -85,B 0,C 180,E1 -16396.409,E2 -16396.409} C_VEL
